KUKA KRL program: ap_15.src, ap_15.dat

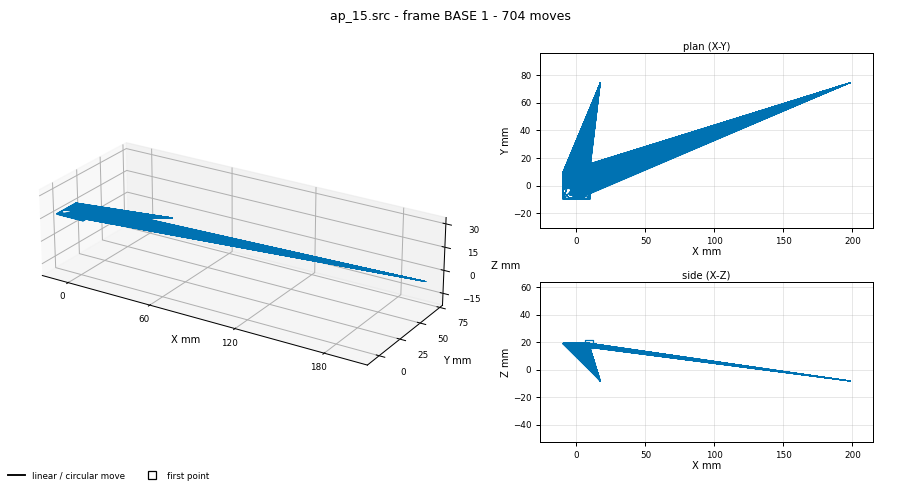
[picture p0: tool path of ap_15.src in frame BASE 1, 704 of 704 moves have a stored position in this frame; points joined in program order, loops and branches not executed]
--- ap_15.src ---
&ACCESS RVP
&REL 65
&PARAM DISKPATH = KRC:\R1\Program
DEF ap_15 ( )
   ;FOLD INI;%{PE}
     ;FOLD BASISTECH INI
       GLOBAL INTERRUPT DECL 3 WHEN $STOPMESS==TRUE DO IR_STOPM ( )
       INTERRUPT ON 3
       BAS (#INITMOV,0 )
     ;ENDFOLD (BASISTECH INI)
     ;FOLD USER INI
       ;Make your modifications here
     ;ENDFOLD (USER INI)
   ;ENDFOLD (INI)

   BAS (#VEL_PTP, 0020.0000)
   BAS (#ACC_PTP, 0020.0000)

   ;-----SET LIN AND ARC MOTION VARIABLES-----
   $VEL.ORI1 = 0350.0000
   $VEL.ORI2 = 0350.0000

   $ACC.CP = 0005.0000
   $ACC.ORI1 = 1000.0000
   $ACC.ORI2 = 1000.0000

   ;-----APPROXIMATION-----
   $APO.CVEL = 0100
   $APO.CPTP = 0100
   $APO.CDIS = 0006.0000
   $APO.CORI = 0090.0000

   BAS (#BASE, 1) ;Positioner
   BAS (#TOOL, 1) ;Vrashatel

   BAS(#VEL_PTP,15)                         ;;Set PTP Axis Velocity
   BAS(#ACC_PTP,50)                         ;;Set PTP Axis Acceleration
   PTP{A1 -92,A2 -133,A3 132,A4 7,A5 50,A6 -10}
   $VEL.CP = 0.060
   LIN  {X 9.039, Y 5.102, Z 18.500, A 0.000, B 0.000, C 0.000} C_DIS
   $VEL.CP = 0.060
   LIN  {X 9.040, Y 9.040, Z 18.500, A 0.000, B 0.000, C 0.000} C_DIS
   $VEL.CP = 0.060
   LIN  {X 9.039, Y 9.039, Z 18.500, A 0.000, B 0.000, C 0.000} C_DIS
   $VEL.CP = 0.060
   LIN  {X 4.069, Y 4.069, Z 18.500, A 0.000, B 0.000, C 0.000} C_DIS
   $VEL.CP = 0.060
   LIN  {X 3.708, Y 3.362, Z 18.500, A 0.000, B 0.000, C 0.000} C_DIS
   $VEL.CP = 0.060
   LIN  {X 9.039, Y -1.968, Z 18.500, A 0.000, B 0.000, C 0.000} C_DIS
   $VEL.CP = 0.060
   LIN  {X 9.039, Y 1.968, Z 18.500, A 0.000, B 0.000, C 0.000} C_DIS
   $VEL.CP = 0.060
   LIN  {X 3.551, Y -3.519, Z 18.500, A 0.000, B 0.000, C 0.000} C_DIS
   $VEL.CP = 0.060
   LIN  {X 0.185, Y -3.520, Z 18.500, A 0.000, B 0.000, C 0.000} C_DIS
   $VEL.CP = 0.060
   LIN  {X 1.313, Y -1.313, Z 18.500, A 0.000, B 0.000, C 0.000} C_DIS
   $VEL.CP = 0.060
   LIN  {X 3.519, Y -3.519, Z 18.500, A 0.000, B 0.000, C 0.000} C_DIS

;FOLD ARCOFF WDAT2 LIN P4 CPDAT2 Tool[1]:cmttorch Base[1]:vrashatel ;%{PE}
  ;FOLD Parameters ;%{h}
    ;Params IlfProvider=kukaroboter.arctech.arcofflin; Kuka.IsGlobalPoint=False; Kuka.PointName=P4; Kuka.BlendingEnabled=False; Kuka.MoveDataName=CPDAT2; Kuka.VelocityPath=0.01; Kuka.CurrentCDSetIndex=0; Kuka.MovementParameterFieldEnabled=True; ArcTech.WdatVarName=WDAT2; ArcTech.Basic=3.4.3.1264
  ;ENDFOLD
  $BWDSTART = FALSE
  LDAT_ACT = LCPDAT2
  FDAT_ACT = FP4
  BAS(#CP_PARAMS, gArcBasVelDefinition)
  SET_CD_PARAMS (0)
  TRIGGER WHEN PATH = ArcGetPath(#ArcOffBefore, WDAT2) DELAY = 0 DO ArcMainNG(#ArcOffBeforeOffStd, WDAT2, WP4) PRIO = -1
  TRIGGER WHEN PATH = ArcGetPath(#OnTheFlyArcOff, WDAT2) DELAY = 0 DO ArcMainNG(#ArcOffMoveStd, WDAT2, WP4) PRIO = -1
  ArcMainNG(#ArcOffBeforeMoveStd, WDAT2, WP4)
  LIN XP4
  ArcMainNG(#ArcOffAfterMoveStd, WDAT2, WP4)
;ENDFOLD
   $VEL.CP = 0.060
   LIN  {X 3.589, Y -3.589, Z 18.500, A 0.000, B 0.000, C 0.000} C_DIS
   $VEL.CP = 0.080
   LIN  {X 4.540, Y -4.052, Z 18.500, A 0.000, B 0.000, C 0.000} C_DIS
   $VEL.CP = 0.080
   LIN  {X 5.072, Y -6.953, Z 18.500, A 0.000, B 0.000, C 0.000} C_DIS

;FOLD ARCON WDAT1 LIN P3 Vel=0.5 m/s CPDAT1 Tool[1]:cmttorch Base[1]:vrashatel ;%{PE}
  ;FOLD Parameters ;%{h}
    ;Params IlfProvider=kukaroboter.arctech.arconlin; Kuka.IsGlobalPoint=False; Kuka.PointName=P3; Kuka.BlendingEnabled=False; Kuka.MoveDataName=CPDAT1; Kuka.VelocityPath=0.5; Kuka.CurrentCDSetIndex=0; Kuka.MovementParameterFieldEnabled=True; ArcTech.WdatVarName=WDAT1; ArcTech.Basic=3.4.3.1264
  ;ENDFOLD
  $BWDSTART = FALSE
  LDAT_ACT = LCPDAT1
  FDAT_ACT = FP3
  BAS(#CP_PARAMS, 0.5)
  SET_CD_PARAMS (0)
  TRIGGER WHEN DISTANCE = 1 DELAY = ArcGetDelay(#PreDefinition, WDAT1) DO ArcMainNG(#PreDefinition, WDAT1, WP3) PRIO = -1
  TRIGGER WHEN PATH = ArcGetPath(#OnTheFlyArcOn, WDAT1) DELAY = ArcGetDelay(#GasPreflow, WDAT1) DO ArcMainNG(#GasPreflow, WDAT1, WP3) PRIO = -1
  TRIGGER WHEN PATH = ArcGetPath(#OnTheFlyArcOn, WDAT1) DELAY = 0 DO ArcMainNG(#ArcOnMoveStd, WDAT1, WP3) PRIO = -1
  ArcMainNG(#ArcOnBeforeMoveStd, WDAT1, WP3)
  LIN XP3
  ArcMainNG(#ArcOnAfterMoveStd, WDAT1, WP3)
;ENDFOLD
   $VEL.CP = 0.060
   LIN  {X 5.071, Y -5.071, Z 18.500, A 0.000, B 0.000, C 0.000} C_DIS
   $VEL.CP = 0.060
   LIN  {X 9.039, Y -9.039, Z 18.500, A 0.000, B 0.000, C 0.000} C_DIS
   $VEL.CP = 0.060
   LIN  {X 9.039, Y -5.102, Z 18.500, A 0.000, B 0.000, C 0.000} C_DIS
   $VEL.CP = 0.060
   LIN  {X 5.102, Y -9.039, Z 18.500, A 0.000, B 0.000, C 0.000} C_DIS
   $VEL.CP = 0.060
   LIN  {X 1.968, Y -9.039, Z 18.500, A 0.000, B 0.000, C 0.000} C_DIS
   $VEL.CP = 0.060
   LIN  {X -0.118, Y -6.952, Z 18.500, A 0.000, B 0.000, C 0.000} C_DIS
   $VEL.CP = 0.060
   LIN  {X 0.118, Y -6.952, Z 18.500, A 0.000, B 0.000, C 0.000} C_DIS
   $VEL.CP = 0.060
   LIN  {X -1.968, Y -9.039, Z 18.500, A 0.000, B 0.000, C 0.000} C_DIS
   $VEL.CP = 0.060
   LIN  {X -5.102, Y -9.039, Z 18.500, A 0.000, B 0.000, C 0.000} C_DIS
   $VEL.CP = 0.060
   LIN  {X -9.039, Y -5.102, Z 18.500, A 0.000, B 0.000, C 0.000} C_DIS
   $VEL.CP = 0.060
   LIN  {X -9.039, Y -9.039, Z 18.500, A 0.000, B 0.000, C 0.000} C_DIS
   $VEL.CP = 0.060
   LIN  {X -3.903, Y -3.903, Z 18.500, A 0.000, B 0.000, C 0.000} C_DIS
   $VEL.CP = 0.060
   LIN  {X -3.655, Y -3.415, Z 18.500, A 0.000, B 0.000, C 0.000} C_DIS
   $VEL.CP = 0.060
   LIN  {X -9.039, Y 1.968, Z 18.500, A 0.000, B 0.000, C 0.000} C_DIS
   $VEL.CP = 0.060
   LIN  {X -9.039, Y -1.968, Z 18.500, A 0.000, B 0.000, C 0.000} C_DIS
   $VEL.CP = 0.060
   LIN  {X -3.226, Y 3.844, Z 18.500, A 0.000, B 0.000, C 0.000} C_DIS
   $VEL.CP = 0.060
   LIN  {X 0.049, Y 3.845, Z 18.500, A 0.000, B 0.000, C 0.000} C_DIS
   $VEL.CP = 0.060
   LIN  {X -1.267, Y 1.267, Z 18.500, A 0.000, B 0.000, C 0.000} C_DIS
   $VEL.CP = 0.060
   LIN  {X -3.844, Y 3.844, Z 18.500, A 0.000, B 0.000, C 0.000} C_DIS
   $VEL.CP = 0.060
   LIN  {X -4.554, Y 3.845, Z 18.500, A 0.000, B 0.000, C 0.000} C_DIS
   $VEL.CP = 0.060
   LIN  {X -4.553, Y 4.553, Z 18.500, A 0.000, B 0.000, C 0.000} C_DIS
   $VEL.CP = 0.060
   LIN  {X -9.039, Y 9.039, Z 18.500, A 0.000, B 0.000, C 0.000} C_DIS
   $VEL.CP = 0.060
   LIN  {X -9.040, Y 9.040, Z 18.500, A 0.000, B 0.000, C 0.000} C_DIS

;FOLD ARCOFF WDAT2 LIN P4 CPDAT2 Tool[1]:cmttorch Base[1]:vrashatel ;%{PE}
  ;FOLD Parameters ;%{h}
    ;Params IlfProvider=kukaroboter.arctech.arcofflin; Kuka.IsGlobalPoint=False; Kuka.PointName=P4; Kuka.BlendingEnabled=False; Kuka.MoveDataName=CPDAT2; Kuka.VelocityPath=0.01; Kuka.CurrentCDSetIndex=0; Kuka.MovementParameterFieldEnabled=True; ArcTech.WdatVarName=WDAT2; ArcTech.Basic=3.4.3.1264
  ;ENDFOLD
  $BWDSTART = FALSE
  LDAT_ACT = LCPDAT2
  FDAT_ACT = FP4
  BAS(#CP_PARAMS, gArcBasVelDefinition)
  SET_CD_PARAMS (0)
  TRIGGER WHEN PATH = ArcGetPath(#ArcOffBefore, WDAT2) DELAY = 0 DO ArcMainNG(#ArcOffBeforeOffStd, WDAT2, WP4) PRIO = -1
  TRIGGER WHEN PATH = ArcGetPath(#OnTheFlyArcOff, WDAT2) DELAY = 0 DO ArcMainNG(#ArcOffMoveStd, WDAT2, WP4) PRIO = -1
  ArcMainNG(#ArcOffBeforeMoveStd, WDAT2, WP4)
  LIN XP4
  ArcMainNG(#ArcOffAfterMoveStd, WDAT2, WP4)
;ENDFOLD
   $VEL.CP = 0.010
   LIN  {X -9.040, Y 9.040, Z 18.700, A 0.000, B 0.000, C 0.000} C_DIS
   $VEL.CP = 0.080
   LIN  {X -9.530, Y 9.530, Z 18.700, A 0.000, B 0.000, C 0.000} C_DIS
   $VEL.CP = 0.080
   LIN  {X -9.800, Y 9.800, Z 18.700, A 0.000, B 0.000, C 0.000} C_DIS

;FOLD ARCON WDAT1 LIN P3 Vel=0.5 m/s CPDAT1 Tool[1]:cmttorch Base[1]:vrashatel ;%{PE}
  ;FOLD Parameters ;%{h}
    ;Params IlfProvider=kukaroboter.arctech.arconlin; Kuka.IsGlobalPoint=False; Kuka.PointName=P3; Kuka.BlendingEnabled=False; Kuka.MoveDataName=CPDAT1; Kuka.VelocityPath=0.5; Kuka.CurrentCDSetIndex=0; Kuka.MovementParameterFieldEnabled=True; ArcTech.WdatVarName=WDAT1; ArcTech.Basic=3.4.3.1264
  ;ENDFOLD
  $BWDSTART = FALSE
  LDAT_ACT = LCPDAT1
  FDAT_ACT = FP3
  BAS(#CP_PARAMS, 0.5)
  SET_CD_PARAMS (0)
  TRIGGER WHEN DISTANCE = 1 DELAY = ArcGetDelay(#PreDefinition, WDAT1) DO ArcMainNG(#PreDefinition, WDAT1, WP3) PRIO = -1
  TRIGGER WHEN PATH = ArcGetPath(#OnTheFlyArcOn, WDAT1) DELAY = ArcGetDelay(#GasPreflow, WDAT1) DO ArcMainNG(#GasPreflow, WDAT1, WP3) PRIO = -1
  TRIGGER WHEN PATH = ArcGetPath(#OnTheFlyArcOn, WDAT1) DELAY = 0 DO ArcMainNG(#ArcOnMoveStd, WDAT1, WP3) PRIO = -1
  ArcMainNG(#ArcOnBeforeMoveStd, WDAT1, WP3)
  LIN XP3
  ArcMainNG(#ArcOnAfterMoveStd, WDAT1, WP3)
;ENDFOLD
   $VEL.CP = 0.025
   LIN  {X -9.800, Y 9.800, Z 18.700, A 0.000, B 0.000, C 0.000} C_DIS
   $VEL.CP = 0.060
   LIN  {X -9.800, Y -9.800, Z 18.700, A 0.000, B 0.000, C 0.000} C_DIS
   $VEL.CP = 0.060
   LIN  {X 9.800, Y -9.800, Z 18.700, A 0.000, B 0.000, C 0.000} C_DIS
   $VEL.CP = 0.060
   LIN  {X 9.800, Y 9.800, Z 18.700, A 0.000, B 0.000, C 0.000} C_DIS
   $VEL.CP = 0.060
   LIN  {X -9.800, Y 9.800, Z 18.700, A 0.000, B 0.000, C 0.000} C_DIS

;FOLD ARCOFF WDAT2 LIN P4 CPDAT2 Tool[1]:cmttorch Base[1]:vrashatel ;%{PE}
  ;FOLD Parameters ;%{h}
    ;Params IlfProvider=kukaroboter.arctech.arcofflin; Kuka.IsGlobalPoint=False; Kuka.PointName=P4; Kuka.BlendingEnabled=False; Kuka.MoveDataName=CPDAT2; Kuka.VelocityPath=0.01; Kuka.CurrentCDSetIndex=0; Kuka.MovementParameterFieldEnabled=True; ArcTech.WdatVarName=WDAT2; ArcTech.Basic=3.4.3.1264
  ;ENDFOLD
  $BWDSTART = FALSE
  LDAT_ACT = LCPDAT2
  FDAT_ACT = FP4
  BAS(#CP_PARAMS, gArcBasVelDefinition)
  SET_CD_PARAMS (0)
  TRIGGER WHEN PATH = ArcGetPath(#ArcOffBefore, WDAT2) DELAY = 0 DO ArcMainNG(#ArcOffBeforeOffStd, WDAT2, WP4) PRIO = -1
  TRIGGER WHEN PATH = ArcGetPath(#OnTheFlyArcOff, WDAT2) DELAY = 0 DO ArcMainNG(#ArcOffMoveStd, WDAT2, WP4) PRIO = -1
  ArcMainNG(#ArcOffBeforeMoveStd, WDAT2, WP4)
  LIN XP4
  ArcMainNG(#ArcOffAfterMoveStd, WDAT2, WP4)
;ENDFOLD
   $VEL.CP = 0.080
   LIN  {X -9.800, Y 9.600, Z 18.700, A 0.000, B 0.000, C 0.000} C_DIS
   $VEL.CP = 0.080
   LIN  {X -9.360, Y 9.360, Z 18.700, A 0.000, B 0.000, C 0.000} C_DIS
   $VEL.CP = 0.080
   LIN  {X -4.094, Y 4.605, Z 18.700, A 0.000, B 0.000, C 0.000} C_DIS
   $VEL.CP = 0.080
   LIN  {X -3.794, Y 4.605, Z 18.700, A 0.000, B 0.000, C 0.000} C_DIS

;FOLD ARCON WDAT1 LIN P3 Vel=0.5 m/s CPDAT1 Tool[1]:cmttorch Base[1]:vrashatel ;%{PE}
  ;FOLD Parameters ;%{h}
    ;Params IlfProvider=kukaroboter.arctech.arconlin; Kuka.IsGlobalPoint=False; Kuka.PointName=P3; Kuka.BlendingEnabled=False; Kuka.MoveDataName=CPDAT1; Kuka.VelocityPath=0.5; Kuka.CurrentCDSetIndex=0; Kuka.MovementParameterFieldEnabled=True; ArcTech.WdatVarName=WDAT1; ArcTech.Basic=3.4.3.1264
  ;ENDFOLD
  $BWDSTART = FALSE
  LDAT_ACT = LCPDAT1
  FDAT_ACT = FP3
  BAS(#CP_PARAMS, 0.5)
  SET_CD_PARAMS (0)
  TRIGGER WHEN DISTANCE = 1 DELAY = ArcGetDelay(#PreDefinition, WDAT1) DO ArcMainNG(#PreDefinition, WDAT1, WP3) PRIO = -1
  TRIGGER WHEN PATH = ArcGetPath(#OnTheFlyArcOn, WDAT1) DELAY = ArcGetDelay(#GasPreflow, WDAT1) DO ArcMainNG(#GasPreflow, WDAT1, WP3) PRIO = -1
  TRIGGER WHEN PATH = ArcGetPath(#OnTheFlyArcOn, WDAT1) DELAY = 0 DO ArcMainNG(#ArcOnMoveStd, WDAT1, WP3) PRIO = -1
  ArcMainNG(#ArcOnBeforeMoveStd, WDAT1, WP3)
  LIN XP3
  ArcMainNG(#ArcOnAfterMoveStd, WDAT1, WP3)
;ENDFOLD
   $VEL.CP = 0.060
   LIN  {X -3.794, Y 6.518, Z 18.700, A 0.000, B 0.000, C 0.000} C_DIS
   $VEL.CP = 0.060
   LIN  {X 4.127, Y 6.518, Z 18.700, A 0.000, B 0.000, C 0.000} C_DIS
   $VEL.CP = 0.060
   LIN  {X 4.127, Y 5.850, Z 18.700, A 0.000, B 0.000, C 0.000} C_DIS
   $VEL.CP = 0.060
   LIN  {X -1.057, Y -4.280, Z 18.700, A 0.000, B 0.000, C 0.000} C_DIS
   $VEL.CP = 0.060
   LIN  {X 4.312, Y -4.280, Z 18.700, A 0.000, B 0.000, C 0.000} C_DIS
   $VEL.CP = 0.060
   LIN  {X 4.312, Y -6.193, Z 18.700, A 0.000, B 0.000, C 0.000} C_DIS
   $VEL.CP = 0.060
   LIN  {X -3.878, Y -6.193, Z 18.700, A 0.000, B 0.000, C 0.000} C_DIS
   $VEL.CP = 0.060
   LIN  {X -3.878, Y -5.525, Z 18.700, A 0.000, B 0.000, C 0.000} C_DIS
   $VEL.CP = 0.060
   LIN  {X 1.290, Y 4.605, Z 18.700, A 0.000, B 0.000, C 0.000} C_DIS
   $VEL.CP = 0.060
   LIN  {X -3.794, Y 4.605, Z 18.700, A 0.000, B 0.000, C 0.000} C_DIS

;FOLD ARCOFF WDAT2 LIN P4 CPDAT2 Tool[1]:cmttorch Base[1]:vrashatel ;%{PE}
  ;FOLD Parameters ;%{h}
    ;Params IlfProvider=kukaroboter.arctech.arcofflin; Kuka.IsGlobalPoint=False; Kuka.PointName=P4; Kuka.BlendingEnabled=False; Kuka.MoveDataName=CPDAT2; Kuka.VelocityPath=0.01; Kuka.CurrentCDSetIndex=0; Kuka.MovementParameterFieldEnabled=True; ArcTech.WdatVarName=WDAT2; ArcTech.Basic=3.4.3.1264
  ;ENDFOLD
  $BWDSTART = FALSE
  LDAT_ACT = LCPDAT2
  FDAT_ACT = FP4
  BAS(#CP_PARAMS, gArcBasVelDefinition)
  SET_CD_PARAMS (0)
  TRIGGER WHEN PATH = ArcGetPath(#ArcOffBefore, WDAT2) DELAY = 0 DO ArcMainNG(#ArcOffBeforeOffStd, WDAT2, WP4) PRIO = -1
  TRIGGER WHEN PATH = ArcGetPath(#OnTheFlyArcOff, WDAT2) DELAY = 0 DO ArcMainNG(#ArcOffMoveStd, WDAT2, WP4) PRIO = -1
  ArcMainNG(#ArcOffBeforeMoveStd, WDAT2, WP4)
  LIN XP4
  ArcMainNG(#ArcOffAfterMoveStd, WDAT2, WP4)
;ENDFOLD
   $VEL.CP = 0.080
   LIN  {X -3.794, Y 4.805, Z 18.700, A 0.000, B 0.000, C 0.000} C_DIS
   $VEL.CP = 0.080
   LIN  {X -4.194, Y 4.205, Z 18.700, A 0.000, B 0.000, C 0.000} C_DIS

;FOLD ARCON WDAT1 LIN P3 Vel=0.5 m/s CPDAT1 Tool[1]:cmttorch Base[1]:vrashatel ;%{PE}
  ;FOLD Parameters ;%{h}
    ;Params IlfProvider=kukaroboter.arctech.arconlin; Kuka.IsGlobalPoint=False; Kuka.PointName=P3; Kuka.BlendingEnabled=False; Kuka.MoveDataName=CPDAT1; Kuka.VelocityPath=0.5; Kuka.CurrentCDSetIndex=0; Kuka.MovementParameterFieldEnabled=True; ArcTech.WdatVarName=WDAT1; ArcTech.Basic=3.4.3.1264
  ;ENDFOLD
  $BWDSTART = FALSE
  LDAT_ACT = LCPDAT1
  FDAT_ACT = FP3
  BAS(#CP_PARAMS, 0.5)
  SET_CD_PARAMS (0)
  TRIGGER WHEN DISTANCE = 1 DELAY = ArcGetDelay(#PreDefinition, WDAT1) DO ArcMainNG(#PreDefinition, WDAT1, WP3) PRIO = -1
  TRIGGER WHEN PATH = ArcGetPath(#OnTheFlyArcOn, WDAT1) DELAY = ArcGetDelay(#GasPreflow, WDAT1) DO ArcMainNG(#GasPreflow, WDAT1, WP3) PRIO = -1
  TRIGGER WHEN PATH = ArcGetPath(#OnTheFlyArcOn, WDAT1) DELAY = 0 DO ArcMainNG(#ArcOnMoveStd, WDAT1, WP3) PRIO = -1
  ArcMainNG(#ArcOnBeforeMoveStd, WDAT1, WP3)
  LIN XP3
  ArcMainNG(#ArcOnAfterMoveStd, WDAT1, WP3)
;ENDFOLD
   $VEL.CP = 0.060
   LIN  {X -4.194, Y 6.918, Z 18.700, A 0.000, B 0.000, C 0.000} C_DIS
   $VEL.CP = 0.060
   LIN  {X 4.527, Y 6.918, Z 18.700, A 0.000, B 0.000, C 0.000} C_DIS
   $VEL.CP = 0.060
   LIN  {X 4.527, Y 5.754, Z 18.700, A 0.000, B 0.000, C 0.000} C_DIS
   $VEL.CP = 0.060
   LIN  {X -0.403, Y -3.880, Z 18.700, A 0.000, B 0.000, C 0.000} C_DIS
   $VEL.CP = 0.060
   LIN  {X 4.712, Y -3.880, Z 18.700, A 0.000, B 0.000, C 0.000} C_DIS
   $VEL.CP = 0.060
   LIN  {X 4.712, Y -6.593, Z 18.700, A 0.000, B 0.000, C 0.000} C_DIS
   $VEL.CP = 0.060
   LIN  {X -4.278, Y -6.593, Z 18.700, A 0.000, B 0.000, C 0.000} C_DIS
   $VEL.CP = 0.060
   LIN  {X -4.278, Y -5.429, Z 18.700, A 0.000, B 0.000, C 0.000} C_DIS
   $VEL.CP = 0.060
   LIN  {X 0.637, Y 4.205, Z 18.700, A 0.000, B 0.000, C 0.000} C_DIS
   $VEL.CP = 0.060
   LIN  {X -4.194, Y 4.205, Z 18.700, A 0.000, B 0.000, C 0.000} C_DIS

;FOLD ARCOFF WDAT2 LIN P4 CPDAT2 Tool[1]:cmttorch Base[1]:vrashatel ;%{PE}
  ;FOLD Parameters ;%{h}
    ;Params IlfProvider=kukaroboter.arctech.arcofflin; Kuka.IsGlobalPoint=False; Kuka.PointName=P4; Kuka.BlendingEnabled=False; Kuka.MoveDataName=CPDAT2; Kuka.VelocityPath=0.01; Kuka.CurrentCDSetIndex=0; Kuka.MovementParameterFieldEnabled=True; ArcTech.WdatVarName=WDAT2; ArcTech.Basic=3.4.3.1264
  ;ENDFOLD
  $BWDSTART = FALSE
  LDAT_ACT = LCPDAT2
  FDAT_ACT = FP4
  BAS(#CP_PARAMS, gArcBasVelDefinition)
  SET_CD_PARAMS (0)
  TRIGGER WHEN PATH = ArcGetPath(#ArcOffBefore, WDAT2) DELAY = 0 DO ArcMainNG(#ArcOffBeforeOffStd, WDAT2, WP4) PRIO = -1
  TRIGGER WHEN PATH = ArcGetPath(#OnTheFlyArcOff, WDAT2) DELAY = 0 DO ArcMainNG(#ArcOffMoveStd, WDAT2, WP4) PRIO = -1
  ArcMainNG(#ArcOffBeforeMoveStd, WDAT2, WP4)
  LIN XP4
  ArcMainNG(#ArcOffAfterMoveStd, WDAT2, WP4)
;ENDFOLD
   $VEL.CP = 0.080
   LIN  {X -9.400, Y 9.400, Z 18.700, A 0.000, B 0.000, C 0.000} C_DIS

;FOLD ARCON WDAT1 LIN P3 Vel=0.5 m/s CPDAT1 Tool[1]:cmttorch Base[1]:vrashatel ;%{PE}
  ;FOLD Parameters ;%{h}
    ;Params IlfProvider=kukaroboter.arctech.arconlin; Kuka.IsGlobalPoint=False; Kuka.PointName=P3; Kuka.BlendingEnabled=False; Kuka.MoveDataName=CPDAT1; Kuka.VelocityPath=0.5; Kuka.CurrentCDSetIndex=0; Kuka.MovementParameterFieldEnabled=True; ArcTech.WdatVarName=WDAT1; ArcTech.Basic=3.4.3.1264
  ;ENDFOLD
  $BWDSTART = FALSE
  LDAT_ACT = LCPDAT1
  FDAT_ACT = FP3
  BAS(#CP_PARAMS, 0.5)
  SET_CD_PARAMS (0)
  TRIGGER WHEN DISTANCE = 1 DELAY = ArcGetDelay(#PreDefinition, WDAT1) DO ArcMainNG(#PreDefinition, WDAT1, WP3) PRIO = -1
  TRIGGER WHEN PATH = ArcGetPath(#OnTheFlyArcOn, WDAT1) DELAY = ArcGetDelay(#GasPreflow, WDAT1) DO ArcMainNG(#GasPreflow, WDAT1, WP3) PRIO = -1
  TRIGGER WHEN PATH = ArcGetPath(#OnTheFlyArcOn, WDAT1) DELAY = 0 DO ArcMainNG(#ArcOnMoveStd, WDAT1, WP3) PRIO = -1
  ArcMainNG(#ArcOnBeforeMoveStd, WDAT1, WP3)
  LIN XP3
  ArcMainNG(#ArcOnAfterMoveStd, WDAT1, WP3)
;ENDFOLD
   $VEL.CP = 0.060
   LIN  {X -9.400, Y -9.400, Z 18.700, A 0.000, B 0.000, C 0.000} C_DIS
   $VEL.CP = 0.060
   LIN  {X 9.400, Y -9.400, Z 18.700, A 0.000, B 0.000, C 0.000} C_DIS
   $VEL.CP = 0.060
   LIN  {X 9.400, Y 9.400, Z 18.700, A 0.000, B 0.000, C 0.000} C_DIS
   $VEL.CP = 0.060
   LIN  {X -9.400, Y 9.400, Z 18.700, A 0.000, B 0.000, C 0.000} C_DIS

;FOLD ARCOFF WDAT2 LIN P4 CPDAT2 Tool[1]:cmttorch Base[1]:vrashatel ;%{PE}
  ;FOLD Parameters ;%{h}
    ;Params IlfProvider=kukaroboter.arctech.arcofflin; Kuka.IsGlobalPoint=False; Kuka.PointName=P4; Kuka.BlendingEnabled=False; Kuka.MoveDataName=CPDAT2; Kuka.VelocityPath=0.01; Kuka.CurrentCDSetIndex=0; Kuka.MovementParameterFieldEnabled=True; ArcTech.WdatVarName=WDAT2; ArcTech.Basic=3.4.3.1264
  ;ENDFOLD
  $BWDSTART = FALSE
  LDAT_ACT = LCPDAT2
  FDAT_ACT = FP4
  BAS(#CP_PARAMS, gArcBasVelDefinition)
  SET_CD_PARAMS (0)
  TRIGGER WHEN PATH = ArcGetPath(#ArcOffBefore, WDAT2) DELAY = 0 DO ArcMainNG(#ArcOffBeforeOffStd, WDAT2, WP4) PRIO = -1
  TRIGGER WHEN PATH = ArcGetPath(#OnTheFlyArcOff, WDAT2) DELAY = 0 DO ArcMainNG(#ArcOffMoveStd, WDAT2, WP4) PRIO = -1
  ArcMainNG(#ArcOffBeforeMoveStd, WDAT2, WP4)
  LIN XP4
  ArcMainNG(#ArcOffAfterMoveStd, WDAT2, WP4)
;ENDFOLD
   $VEL.CP = 0.080
   LIN  {X -9.040, Y 9.040, Z 18.700, A 0.000, B 0.000, C 0.000} C_DIS

;FOLD ARCON WDAT1 LIN P3 Vel=0.5 m/s CPDAT1 Tool[1]:cmttorch Base[1]:vrashatel ;%{PE}
  ;FOLD Parameters ;%{h}
    ;Params IlfProvider=kukaroboter.arctech.arconlin; Kuka.IsGlobalPoint=False; Kuka.PointName=P3; Kuka.BlendingEnabled=False; Kuka.MoveDataName=CPDAT1; Kuka.VelocityPath=0.5; Kuka.CurrentCDSetIndex=0; Kuka.MovementParameterFieldEnabled=True; ArcTech.WdatVarName=WDAT1; ArcTech.Basic=3.4.3.1264
  ;ENDFOLD
  $BWDSTART = FALSE
  LDAT_ACT = LCPDAT1
  FDAT_ACT = FP3
  BAS(#CP_PARAMS, 0.5)
  SET_CD_PARAMS (0)
  TRIGGER WHEN DISTANCE = 1 DELAY = ArcGetDelay(#PreDefinition, WDAT1) DO ArcMainNG(#PreDefinition, WDAT1, WP3) PRIO = -1
  TRIGGER WHEN PATH = ArcGetPath(#OnTheFlyArcOn, WDAT1) DELAY = ArcGetDelay(#GasPreflow, WDAT1) DO ArcMainNG(#GasPreflow, WDAT1, WP3) PRIO = -1
  TRIGGER WHEN PATH = ArcGetPath(#OnTheFlyArcOn, WDAT1) DELAY = 0 DO ArcMainNG(#ArcOnMoveStd, WDAT1, WP3) PRIO = -1
  ArcMainNG(#ArcOnBeforeMoveStd, WDAT1, WP3)
  LIN XP3
  ArcMainNG(#ArcOnAfterMoveStd, WDAT1, WP3)
;ENDFOLD
   $VEL.CP = 0.060
   LIN  {X -9.039, Y 5.102, Z 18.700, A 0.000, B 0.000, C 0.000} C_DIS
   $VEL.CP = 0.060
   LIN  {X -5.102, Y 9.039, Z 18.700, A 0.000, B 0.000, C 0.000} C_DIS
   $VEL.CP = 0.060
   LIN  {X -1.968, Y 9.039, Z 18.700, A 0.000, B 0.000, C 0.000} C_DIS
   $VEL.CP = 0.060
   LIN  {X -0.205, Y 7.276, Z 18.700, A 0.000, B 0.000, C 0.000} C_DIS
   $VEL.CP = 0.060
   LIN  {X 0.206, Y 7.277, Z 18.700, A 0.000, B 0.000, C 0.000} C_DIS
   $VEL.CP = 0.060
   LIN  {X 1.968, Y 9.039, Z 18.700, A 0.000, B 0.000, C 0.000} C_DIS
   $VEL.CP = 0.060
   LIN  {X 5.102, Y 9.039, Z 18.700, A 0.000, B 0.000, C 0.000} C_DIS
   $VEL.CP = 0.060
   LIN  {X 9.039, Y 5.102, Z 18.700, A 0.000, B 0.000, C 0.000} C_DIS
   $VEL.CP = 0.060
   LIN  {X 9.040, Y 9.040, Z 18.700, A 0.000, B 0.000, C 0.000} C_DIS
   $VEL.CP = 0.060
   LIN  {X 9.039, Y 9.039, Z 18.700, A 0.000, B 0.000, C 0.000} C_DIS
   $VEL.CP = 0.060
   LIN  {X 4.069, Y 4.069, Z 18.700, A 0.000, B 0.000, C 0.000} C_DIS
   $VEL.CP = 0.060
   LIN  {X 3.708, Y 3.362, Z 18.700, A 0.000, B 0.000, C 0.000} C_DIS
   $VEL.CP = 0.060
   LIN  {X 9.039, Y -1.968, Z 18.700, A 0.000, B 0.000, C 0.000} C_DIS
   $VEL.CP = 0.060
   LIN  {X 9.039, Y 1.968, Z 18.700, A 0.000, B 0.000, C 0.000} C_DIS
   $VEL.CP = 0.060
   LIN  {X 3.551, Y -3.519, Z 18.700, A 0.000, B 0.000, C 0.000} C_DIS
   $VEL.CP = 0.060
   LIN  {X 0.185, Y -3.520, Z 18.700, A 0.000, B 0.000, C 0.000} C_DIS
   $VEL.CP = 0.060
   LIN  {X 1.313, Y -1.313, Z 18.700, A 0.000, B 0.000, C 0.000} C_DIS
   $VEL.CP = 0.060
   LIN  {X 3.519, Y -3.519, Z 18.700, A 0.000, B 0.000, C 0.000} C_DIS

;FOLD ARCOFF WDAT2 LIN P4 CPDAT2 Tool[1]:cmttorch Base[1]:vrashatel ;%{PE}
  ;FOLD Parameters ;%{h}
    ;Params IlfProvider=kukaroboter.arctech.arcofflin; Kuka.IsGlobalPoint=False; Kuka.PointName=P4; Kuka.BlendingEnabled=False; Kuka.MoveDataName=CPDAT2; Kuka.VelocityPath=0.01; Kuka.CurrentCDSetIndex=0; Kuka.MovementParameterFieldEnabled=True; ArcTech.WdatVarName=WDAT2; ArcTech.Basic=3.4.3.1264
  ;ENDFOLD
  $BWDSTART = FALSE
  LDAT_ACT = LCPDAT2
  FDAT_ACT = FP4
  BAS(#CP_PARAMS, gArcBasVelDefinition)
  SET_CD_PARAMS (0)
  TRIGGER WHEN PATH = ArcGetPath(#ArcOffBefore, WDAT2) DELAY = 0 DO ArcMainNG(#ArcOffBeforeOffStd, WDAT2, WP4) PRIO = -1
  TRIGGER WHEN PATH = ArcGetPath(#OnTheFlyArcOff, WDAT2) DELAY = 0 DO ArcMainNG(#ArcOffMoveStd, WDAT2, WP4) PRIO = -1
  ArcMainNG(#ArcOffBeforeMoveStd, WDAT2, WP4)
  LIN XP4
  ArcMainNG(#ArcOffAfterMoveStd, WDAT2, WP4)
;ENDFOLD
   $VEL.CP = 0.060
   LIN  {X 3.589, Y -3.589, Z 18.700, A 0.000, B 0.000, C 0.000} C_DIS
   $VEL.CP = 0.080
   LIN  {X 4.540, Y -4.052, Z 18.700, A 0.000, B 0.000, C 0.000} C_DIS
   $VEL.CP = 0.080
   LIN  {X 5.072, Y -6.953, Z 18.700, A 0.000, B 0.000, C 0.000} C_DIS

;FOLD ARCON WDAT1 LIN P3 Vel=0.5 m/s CPDAT1 Tool[1]:cmttorch Base[1]:vrashatel ;%{PE}
  ;FOLD Parameters ;%{h}
    ;Params IlfProvider=kukaroboter.arctech.arconlin; Kuka.IsGlobalPoint=False; Kuka.PointName=P3; Kuka.BlendingEnabled=False; Kuka.MoveDataName=CPDAT1; Kuka.VelocityPath=0.5; Kuka.CurrentCDSetIndex=0; Kuka.MovementParameterFieldEnabled=True; ArcTech.WdatVarName=WDAT1; ArcTech.Basic=3.4.3.1264
  ;ENDFOLD
  $BWDSTART = FALSE
  LDAT_ACT = LCPDAT1
  FDAT_ACT = FP3
  BAS(#CP_PARAMS, 0.5)
  SET_CD_PARAMS (0)
  TRIGGER WHEN DISTANCE = 1 DELAY = ArcGetDelay(#PreDefinition, WDAT1) DO ArcMainNG(#PreDefinition, WDAT1, WP3) PRIO = -1
  TRIGGER WHEN PATH = ArcGetPath(#OnTheFlyArcOn, WDAT1) DELAY = ArcGetDelay(#GasPreflow, WDAT1) DO ArcMainNG(#GasPreflow, WDAT1, WP3) PRIO = -1
  TRIGGER WHEN PATH = ArcGetPath(#OnTheFlyArcOn, WDAT1) DELAY = 0 DO ArcMainNG(#ArcOnMoveStd, WDAT1, WP3) PRIO = -1
  ArcMainNG(#ArcOnBeforeMoveStd, WDAT1, WP3)
  LIN XP3
  ArcMainNG(#ArcOnAfterMoveStd, WDAT1, WP3)
;ENDFOLD
   $VEL.CP = 0.060
   LIN  {X 5.071, Y -5.071, Z 18.700, A 0.000, B 0.000, C 0.000} C_DIS
   $VEL.CP = 0.060
   LIN  {X 9.039, Y -9.039, Z 18.700, A 0.000, B 0.000, C 0.000} C_DIS
   $VEL.CP = 0.060
   LIN  {X 9.039, Y -5.102, Z 18.700, A 0.000, B 0.000, C 0.000} C_DIS
   $VEL.CP = 0.060
   LIN  {X 5.102, Y -9.039, Z 18.700, A 0.000, B 0.000, C 0.000} C_DIS
   $VEL.CP = 0.060
   LIN  {X 1.968, Y -9.039, Z 18.700, A 0.000, B 0.000, C 0.000} C_DIS
   $VEL.CP = 0.060
   LIN  {X -0.118, Y -6.952, Z 18.700, A 0.000, B 0.000, C 0.000} C_DIS
   $VEL.CP = 0.060
   LIN  {X 0.118, Y -6.952, Z 18.700, A 0.000, B 0.000, C 0.000} C_DIS
   $VEL.CP = 0.060
   LIN  {X -1.968, Y -9.039, Z 18.700, A 0.000, B 0.000, C 0.000} C_DIS
   $VEL.CP = 0.060
   LIN  {X -5.102, Y -9.039, Z 18.700, A 0.000, B 0.000, C 0.000} C_DIS
   $VEL.CP = 0.060
   LIN  {X -9.039, Y -5.102, Z 18.700, A 0.000, B 0.000, C 0.000} C_DIS
   $VEL.CP = 0.060
   LIN  {X -9.039, Y -9.039, Z 18.700, A 0.000, B 0.000, C 0.000} C_DIS
   $VEL.CP = 0.060
   LIN  {X -3.903, Y -3.903, Z 18.700, A 0.000, B 0.000, C 0.000} C_DIS
   $VEL.CP = 0.060
   LIN  {X -3.655, Y -3.415, Z 18.700, A 0.000, B 0.000, C 0.000} C_DIS
   $VEL.CP = 0.060
   LIN  {X -9.039, Y 1.968, Z 18.700, A 0.000, B 0.000, C 0.000} C_DIS
   $VEL.CP = 0.060
   LIN  {X -9.039, Y -1.968, Z 18.700, A 0.000, B 0.000, C 0.000} C_DIS
   $VEL.CP = 0.060
   LIN  {X -3.226, Y 3.844, Z 18.700, A 0.000, B 0.000, C 0.000} C_DIS
   $VEL.CP = 0.060
   LIN  {X 0.049, Y 3.845, Z 18.700, A 0.000, B 0.000, C 0.000} C_DIS
   $VEL.CP = 0.060
   LIN  {X -1.267, Y 1.267, Z 18.700, A 0.000, B 0.000, C 0.000} C_DIS
   $VEL.CP = 0.060
   LIN  {X -3.844, Y 3.844, Z 18.700, A 0.000, B 0.000, C 0.000} C_DIS
   $VEL.CP = 0.060
   LIN  {X -4.554, Y 3.845, Z 18.700, A 0.000, B 0.000, C 0.000} C_DIS
   $VEL.CP = 0.060
   LIN  {X -4.553, Y 4.553, Z 18.700, A 0.000, B 0.000, C 0.000} C_DIS
   $VEL.CP = 0.060
   LIN  {X -9.039, Y 9.039, Z 18.700, A 0.000, B 0.000, C 0.000} C_DIS
   $VEL.CP = 0.060
   LIN  {X -9.040, Y 9.040, Z 18.700, A 0.000, B 0.000, C 0.000} C_DIS

;FOLD ARCOFF WDAT2 LIN P4 CPDAT2 Tool[1]:cmttorch Base[1]:vrashatel ;%{PE}
  ;FOLD Parameters ;%{h}
    ;Params IlfProvider=kukaroboter.arctech.arcofflin; Kuka.IsGlobalPoint=False; Kuka.PointName=P4; Kuka.BlendingEnabled=False; Kuka.MoveDataName=CPDAT2; Kuka.VelocityPath=0.01; Kuka.CurrentCDSetIndex=0; Kuka.MovementParameterFieldEnabled=True; ArcTech.WdatVarName=WDAT2; ArcTech.Basic=3.4.3.1264
  ;ENDFOLD
  $BWDSTART = FALSE
  LDAT_ACT = LCPDAT2
  FDAT_ACT = FP4
  BAS(#CP_PARAMS, gArcBasVelDefinition)
  SET_CD_PARAMS (0)
  TRIGGER WHEN PATH = ArcGetPath(#ArcOffBefore, WDAT2) DELAY = 0 DO ArcMainNG(#ArcOffBeforeOffStd, WDAT2, WP4) PRIO = -1
  TRIGGER WHEN PATH = ArcGetPath(#OnTheFlyArcOff, WDAT2) DELAY = 0 DO ArcMainNG(#ArcOffMoveStd, WDAT2, WP4) PRIO = -1
  ArcMainNG(#ArcOffBeforeMoveStd, WDAT2, WP4)
  LIN XP4
  ArcMainNG(#ArcOffAfterMoveStd, WDAT2, WP4)
;ENDFOLD
   $VEL.CP = 0.010
   LIN  {X -9.040, Y 9.040, Z 18.900, A 0.000, B 0.000, C 0.000} C_DIS
   $VEL.CP = 0.080
   LIN  {X -9.530, Y 9.530, Z 18.900, A 0.000, B 0.000, C 0.000} C_DIS
   $VEL.CP = 0.080
   LIN  {X -9.800, Y 9.800, Z 18.900, A 0.000, B 0.000, C 0.000} C_DIS

;FOLD ARCON WDAT1 LIN P3 Vel=0.5 m/s CPDAT1 Tool[1]:cmttorch Base[1]:vrashatel ;%{PE}
  ;FOLD Parameters ;%{h}
    ;Params IlfProvider=kukaroboter.arctech.arconlin; Kuka.IsGlobalPoint=False; Kuka.PointName=P3; Kuka.BlendingEnabled=False; Kuka.MoveDataName=CPDAT1; Kuka.VelocityPath=0.5; Kuka.CurrentCDSetIndex=0; Kuka.MovementParameterFieldEnabled=True; ArcTech.WdatVarName=WDAT1; ArcTech.Basic=3.4.3.1264
  ;ENDFOLD
  $BWDSTART = FALSE
  LDAT_ACT = LCPDAT1
  FDAT_ACT = FP3
  BAS(#CP_PARAMS, 0.5)
  SET_CD_PARAMS (0)
  TRIGGER WHEN DISTANCE = 1 DELAY = ArcGetDelay(#PreDefinition, WDAT1) DO ArcMainNG(#PreDefinition, WDAT1, WP3) PRIO = -1
  TRIGGER WHEN PATH = ArcGetPath(#OnTheFlyArcOn, WDAT1) DELAY = ArcGetDelay(#GasPreflow, WDAT1) DO ArcMainNG(#GasPreflow, WDAT1, WP3) PRIO = -1
  TRIGGER WHEN PATH = ArcGetPath(#OnTheFlyArcOn, WDAT1) DELAY = 0 DO ArcMainNG(#ArcOnMoveStd, WDAT1, WP3) PRIO = -1
  ArcMainNG(#ArcOnBeforeMoveStd, WDAT1, WP3)
  LIN XP3
  ArcMainNG(#ArcOnAfterMoveStd, WDAT1, WP3)
;ENDFOLD
   $VEL.CP = 0.025
   LIN  {X -9.800, Y 9.800, Z 18.900, A 0.000, B 0.000, C 0.000} C_DIS
   $VEL.CP = 0.060
   LIN  {X -9.800, Y -9.800, Z 18.900, A 0.000, B 0.000, C 0.000} C_DIS
   $VEL.CP = 0.060
   LIN  {X 9.800, Y -9.800, Z 18.900, A 0.000, B 0.000, C 0.000} C_DIS
   $VEL.CP = 0.060
   LIN  {X 9.800, Y 9.800, Z 18.900, A 0.000, B 0.000, C 0.000} C_DIS
   $VEL.CP = 0.060
   LIN  {X -9.800, Y 9.800, Z 18.900, A 0.000, B 0.000, C 0.000} C_DIS

;FOLD ARCOFF WDAT2 LIN P4 CPDAT2 Tool[1]:cmttorch Base[1]:vrashatel ;%{PE}
  ;FOLD Parameters ;%{h}
    ;Params IlfProvider=kukaroboter.arctech.arcofflin; Kuka.IsGlobalPoint=False; Kuka.PointName=P4; Kuka.BlendingEnabled=False; Kuka.MoveDataName=CPDAT2; Kuka.VelocityPath=0.01; Kuka.CurrentCDSetIndex=0; Kuka.MovementParameterFieldEnabled=True; ArcTech.WdatVarName=WDAT2; ArcTech.Basic=3.4.3.1264
  ;ENDFOLD
  $BWDSTART = FALSE
  LDAT_ACT = LCPDAT2
  FDAT_ACT = FP4
  BAS(#CP_PARAMS, gArcBasVelDefinition)
  SET_CD_PARAMS (0)
  TRIGGER WHEN PATH = ArcGetPath(#ArcOffBefore, WDAT2) DELAY = 0 DO ArcMainNG(#ArcOffBeforeOffStd, WDAT2, WP4) PRIO = -1
  TRIGGER WHEN PATH = ArcGetPath(#OnTheFlyArcOff, WDAT2) DELAY = 0 DO ArcMainNG(#ArcOffMoveStd, WDAT2, WP4) PRIO = -1
  ArcMainNG(#ArcOffBeforeMoveStd, WDAT2, WP4)
  LIN XP4
  ArcMainNG(#ArcOffAfterMoveStd, WDAT2, WP4)
;ENDFOLD
   $VEL.CP = 0.080
   LIN  {X -9.800, Y 9.600, Z 18.900, A 0.000, B 0.000, C 0.000} C_DIS
   $VEL.CP = 0.080
   LIN  {X -9.360, Y 9.360, Z 18.900, A 0.000, B 0.000, C 0.000} C_DIS
   $VEL.CP = 0.080
   LIN  {X -4.094, Y 4.605, Z 18.900, A 0.000, B 0.000, C 0.000} C_DIS
   $VEL.CP = 0.080
   LIN  {X -3.794, Y 4.605, Z 18.900, A 0.000, B 0.000, C 0.000} C_DIS

;FOLD ARCON WDAT1 LIN P3 Vel=0.5 m/s CPDAT1 Tool[1]:cmttorch Base[1]:vrashatel ;%{PE}
  ;FOLD Parameters ;%{h}
    ;Params IlfProvider=kukaroboter.arctech.arconlin; Kuka.IsGlobalPoint=False; Kuka.PointName=P3; Kuka.BlendingEnabled=False; Kuka.MoveDataName=CPDAT1; Kuka.VelocityPath=0.5; Kuka.CurrentCDSetIndex=0; Kuka.MovementParameterFieldEnabled=True; ArcTech.WdatVarName=WDAT1; ArcTech.Basic=3.4.3.1264
  ;ENDFOLD
  $BWDSTART = FALSE
  LDAT_ACT = LCPDAT1
  FDAT_ACT = FP3
  BAS(#CP_PARAMS, 0.5)
  SET_CD_PARAMS (0)
  TRIGGER WHEN DISTANCE = 1 DELAY = ArcGetDelay(#PreDefinition, WDAT1) DO ArcMainNG(#PreDefinition, WDAT1, WP3) PRIO = -1
  TRIGGER WHEN PATH = ArcGetPath(#OnTheFlyArcOn, WDAT1) DELAY = ArcGetDelay(#GasPreflow, WDAT1) DO ArcMainNG(#GasPreflow, WDAT1, WP3) PRIO = -1
  TRIGGER WHEN PATH = ArcGetPath(#OnTheFlyArcOn, WDAT1) DELAY = 0 DO ArcMainNG(#ArcOnMoveStd, WDAT1, WP3) PRIO = -1
  ArcMainNG(#ArcOnBeforeMoveStd, WDAT1, WP3)
  LIN XP3
  ArcMainNG(#ArcOnAfterMoveStd, WDAT1, WP3)
;ENDFOLD
   $VEL.CP = 0.060
   LIN  {X -3.794, Y 6.518, Z 18.900, A 0.000, B 0.000, C 0.000} C_DIS
   $VEL.CP = 0.060
   LIN  {X 4.127, Y 6.518, Z 18.900, A 0.000, B 0.000, C 0.000} C_DIS
   $VEL.CP = 0.060
   LIN  {X 4.127, Y 5.850, Z 18.900, A 0.000, B 0.000, C 0.000} C_DIS
   $VEL.CP = 0.060
   LIN  {X -1.057, Y -4.280, Z 18.900, A 0.000, B 0.000, C 0.000} C_DIS
   $VEL.CP = 0.060
   LIN  {X 4.312, Y -4.280, Z 18.900, A 0.000, B 0.000, C 0.000} C_DIS
   $VEL.CP = 0.060
   LIN  {X 4.312, Y -6.193, Z 18.900, A 0.000, B 0.000, C 0.000} C_DIS
   $VEL.CP = 0.060
   LIN  {X -3.878, Y -6.193, Z 18.900, A 0.000, B 0.000, C 0.000} C_DIS
   $VEL.CP = 0.060
   LIN  {X -3.878, Y -5.525, Z 18.900, A 0.000, B 0.000, C 0.000} C_DIS
   $VEL.CP = 0.060
   LIN  {X 1.290, Y 4.605, Z 18.900, A 0.000, B 0.000, C 0.000} C_DIS
   $VEL.CP = 0.060
   LIN  {X -3.794, Y 4.605, Z 18.900, A 0.000, B 0.000, C 0.000} C_DIS

;FOLD ARCOFF WDAT2 LIN P4 CPDAT2 Tool[1]:cmttorch Base[1]:vrashatel ;%{PE}
  ;FOLD Parameters ;%{h}
    ;Params IlfProvider=kukaroboter.arctech.arcofflin; Kuka.IsGlobalPoint=False; Kuka.PointName=P4; Kuka.BlendingEnabled=False; Kuka.MoveDataName=CPDAT2; Kuka.VelocityPath=0.01; Kuka.CurrentCDSetIndex=0; Kuka.MovementParameterFieldEnabled=True; ArcTech.WdatVarName=WDAT2; ArcTech.Basic=3.4.3.1264
  ;ENDFOLD
  $BWDSTART = FALSE
  LDAT_ACT = LCPDAT2
  FDAT_ACT = FP4
  BAS(#CP_PARAMS, gArcBasVelDefinition)
  SET_CD_PARAMS (0)
  TRIGGER WHEN PATH = ArcGetPath(#ArcOffBefore, WDAT2) DELAY = 0 DO ArcMainNG(#ArcOffBeforeOffStd, WDAT2, WP4) PRIO = -1
  TRIGGER WHEN PATH = ArcGetPath(#OnTheFlyArcOff, WDAT2) DELAY = 0 DO ArcMainNG(#ArcOffMoveStd, WDAT2, WP4) PRIO = -1
  ArcMainNG(#ArcOffBeforeMoveStd, WDAT2, WP4)
  LIN XP4
  ArcMainNG(#ArcOffAfterMoveStd, WDAT2, WP4)
;ENDFOLD
   $VEL.CP = 0.080
   LIN  {X -3.794, Y 4.805, Z 18.900, A 0.000, B 0.000, C 0.000} C_DIS
   $VEL.CP = 0.080
   LIN  {X -4.194, Y 4.205, Z 18.900, A 0.000, B 0.000, C 0.000} C_DIS

;FOLD ARCON WDAT1 LIN P3 Vel=0.5 m/s CPDAT1 Tool[1]:cmttorch Base[1]:vrashatel ;%{PE}
  ;FOLD Parameters ;%{h}
    ;Params IlfProvider=kukaroboter.arctech.arconlin; Kuka.IsGlobalPoint=False; Kuka.PointName=P3; Kuka.BlendingEnabled=False; Kuka.MoveDataName=CPDAT1; Kuka.VelocityPath=0.5; Kuka.CurrentCDSetIndex=0; Kuka.MovementParameterFieldEnabled=True; ArcTech.WdatVarName=WDAT1; ArcTech.Basic=3.4.3.1264
  ;ENDFOLD
  $BWDSTART = FALSE
  LDAT_ACT = LCPDAT1
  FDAT_ACT = FP3
  BAS(#CP_PARAMS, 0.5)
  SET_CD_PARAMS (0)
  TRIGGER WHEN DISTANCE = 1 DELAY = ArcGetDelay(#PreDefinition, WDAT1) DO ArcMainNG(#PreDefinition, WDAT1, WP3) PRIO = -1
  TRIGGER WHEN PATH = ArcGetPath(#OnTheFlyArcOn, WDAT1) DELAY = ArcGetDelay(#GasPreflow, WDAT1) DO ArcMainNG(#GasPreflow, WDAT1, WP3) PRIO = -1
  TRIGGER WHEN PATH = ArcGetPath(#OnTheFlyArcOn, WDAT1) DELAY = 0 DO ArcMainNG(#ArcOnMoveStd, WDAT1, WP3) PRIO = -1
  ArcMainNG(#ArcOnBeforeMoveStd, WDAT1, WP3)
  LIN XP3
  ArcMainNG(#ArcOnAfterMoveStd, WDAT1, WP3)
;ENDFOLD
   $VEL.CP = 0.060
   LIN  {X -4.194, Y 6.918, Z 18.900, A 0.000, B 0.000, C 0.000} C_DIS
   $VEL.CP = 0.060
   LIN  {X 4.527, Y 6.918, Z 18.900, A 0.000, B 0.000, C 0.000} C_DIS
   $VEL.CP = 0.060
   LIN  {X 4.527, Y 5.754, Z 18.900, A 0.000, B 0.000, C 0.000} C_DIS
   $VEL.CP = 0.060
   LIN  {X -0.403, Y -3.880, Z 18.900, A 0.000, B 0.000, C 0.000} C_DIS
   $VEL.CP = 0.060
   LIN  {X 4.712, Y -3.880, Z 18.900, A 0.000, B 0.000, C 0.000} C_DIS
   $VEL.CP = 0.060
   LIN  {X 4.712, Y -6.593, Z 18.900, A 0.000, B 0.000, C 0.000} C_DIS
   $VEL.CP = 0.060
   LIN  {X -4.278, Y -6.593, Z 18.900, A 0.000, B 0.000, C 0.000} C_DIS
   $VEL.CP = 0.060
   LIN  {X -4.278, Y -5.429, Z 18.900, A 0.000, B 0.000, C 0.000} C_DIS
   $VEL.CP = 0.060
   LIN  {X 0.637, Y 4.205, Z 18.900, A 0.000, B 0.000, C 0.000} C_DIS
   $VEL.CP = 0.060
   LIN  {X -4.194, Y 4.205, Z 18.900, A 0.000, B 0.000, C 0.000} C_DIS

;FOLD ARCOFF WDAT2 LIN P4 CPDAT2 Tool[1]:cmttorch Base[1]:vrashatel ;%{PE}
  ;FOLD Parameters ;%{h}
    ;Params IlfProvider=kukaroboter.arctech.arcofflin; Kuka.IsGlobalPoint=False; Kuka.PointName=P4; Kuka.BlendingEnabled=False; Kuka.MoveDataName=CPDAT2; Kuka.VelocityPath=0.01; Kuka.CurrentCDSetIndex=0; Kuka.MovementParameterFieldEnabled=True; ArcTech.WdatVarName=WDAT2; ArcTech.Basic=3.4.3.1264
  ;ENDFOLD
  $BWDSTART = FALSE
  LDAT_ACT = LCPDAT2
  FDAT_ACT = FP4
  BAS(#CP_PARAMS, gArcBasVelDefinition)
  SET_CD_PARAMS (0)
  TRIGGER WHEN PATH = ArcGetPath(#ArcOffBefore, WDAT2) DELAY = 0 DO ArcMainNG(#ArcOffBeforeOffStd, WDAT2, WP4) PRIO = -1
  TRIGGER WHEN PATH = ArcGetPath(#OnTheFlyArcOff, WDAT2) DELAY = 0 DO ArcMainNG(#ArcOffMoveStd, WDAT2, WP4) PRIO = -1
  ArcMainNG(#ArcOffBeforeMoveStd, WDAT2, WP4)
  LIN XP4
  ArcMainNG(#ArcOffAfterMoveStd, WDAT2, WP4)
;ENDFOLD
   $VEL.CP = 0.080
   LIN  {X -9.400, Y 9.400, Z 18.900, A 0.000, B 0.000, C 0.000} C_DIS

;FOLD ARCON WDAT1 LIN P3 Vel=0.5 m/s CPDAT1 Tool[1]:cmttorch Base[1]:vrashatel ;%{PE}
  ;FOLD Parameters ;%{h}
    ;Params IlfProvider=kukaroboter.arctech.arconlin; Kuka.IsGlobalPoint=False; Kuka.PointName=P3; Kuka.BlendingEnabled=False; Kuka.MoveDataName=CPDAT1; Kuka.VelocityPath=0.5; Kuka.CurrentCDSetIndex=0; Kuka.MovementParameterFieldEnabled=True; ArcTech.WdatVarName=WDAT1; ArcTech.Basic=3.4.3.1264
  ;ENDFOLD
  $BWDSTART = FALSE
  LDAT_ACT = LCPDAT1
  FDAT_ACT = FP3
  BAS(#CP_PARAMS, 0.5)
  SET_CD_PARAMS (0)
  TRIGGER WHEN DISTANCE = 1 DELAY = ArcGetDelay(#PreDefinition, WDAT1) DO ArcMainNG(#PreDefinition, WDAT1, WP3) PRIO = -1
  TRIGGER WHEN PATH = ArcGetPath(#OnTheFlyArcOn, WDAT1) DELAY = ArcGetDelay(#GasPreflow, WDAT1) DO ArcMainNG(#GasPreflow, WDAT1, WP3) PRIO = -1
  TRIGGER WHEN PATH = ArcGetPath(#OnTheFlyArcOn, WDAT1) DELAY = 0 DO ArcMainNG(#ArcOnMoveStd, WDAT1, WP3) PRIO = -1
  ArcMainNG(#ArcOnBeforeMoveStd, WDAT1, WP3)
  LIN XP3
  ArcMainNG(#ArcOnAfterMoveStd, WDAT1, WP3)
;ENDFOLD
   $VEL.CP = 0.060
   LIN  {X -9.400, Y -9.400, Z 18.900, A 0.000, B 0.000, C 0.000} C_DIS
   $VEL.CP = 0.060
   LIN  {X 9.400, Y -9.400, Z 18.900, A 0.000, B 0.000, C 0.000} C_DIS
   $VEL.CP = 0.060
   LIN  {X 9.400, Y 9.400, Z 18.900, A 0.000, B 0.000, C 0.000} C_DIS
   $VEL.CP = 0.060
   LIN  {X -9.400, Y 9.400, Z 18.900, A 0.000, B 0.000, C 0.000} C_DIS

;FOLD ARCOFF WDAT2 LIN P4 CPDAT2 Tool[1]:cmttorch Base[1]:vrashatel ;%{PE}
  ;FOLD Parameters ;%{h}
    ;Params IlfProvider=kukaroboter.arctech.arcofflin; Kuka.IsGlobalPoint=False; Kuka.PointName=P4; Kuka.BlendingEnabled=False; Kuka.MoveDataName=CPDAT2; Kuka.VelocityPath=0.01; Kuka.CurrentCDSetIndex=0; Kuka.MovementParameterFieldEnabled=True; ArcTech.WdatVarName=WDAT2; ArcTech.Basic=3.4.3.1264
  ;ENDFOLD
  $BWDSTART = FALSE
  LDAT_ACT = LCPDAT2
  FDAT_ACT = FP4
  BAS(#CP_PARAMS, gArcBasVelDefinition)
  SET_CD_PARAMS (0)
  TRIGGER WHEN PATH = ArcGetPath(#ArcOffBefore, WDAT2) DELAY = 0 DO ArcMainNG(#ArcOffBeforeOffStd, WDAT2, WP4) PRIO = -1
  TRIGGER WHEN PATH = ArcGetPath(#OnTheFlyArcOff, WDAT2) DELAY = 0 DO ArcMainNG(#ArcOffMoveStd, WDAT2, WP4) PRIO = -1
  ArcMainNG(#ArcOffBeforeMoveStd, WDAT2, WP4)
  LIN XP4
  ArcMainNG(#ArcOffAfterMoveStd, WDAT2, WP4)
;ENDFOLD
   $VEL.CP = 0.080
   LIN  {X -9.040, Y 9.040, Z 18.900, A 0.000, B 0.000, C 0.000} C_DIS

;FOLD ARCON WDAT1 LIN P3 Vel=0.5 m/s CPDAT1 Tool[1]:cmttorch Base[1]:vrashatel ;%{PE}
  ;FOLD Parameters ;%{h}
    ;Params IlfProvider=kukaroboter.arctech.arconlin; Kuka.IsGlobalPoint=False; Kuka.PointName=P3; Kuka.BlendingEnabled=False; Kuka.MoveDataName=CPDAT1; Kuka.VelocityPath=0.5; Kuka.CurrentCDSetIndex=0; Kuka.MovementParameterFieldEnabled=True; ArcTech.WdatVarName=WDAT1; ArcTech.Basic=3.4.3.1264
  ;ENDFOLD
  $BWDSTART = FALSE
  LDAT_ACT = LCPDAT1
  FDAT_ACT = FP3
  BAS(#CP_PARAMS, 0.5)
  SET_CD_PARAMS (0)
  TRIGGER WHEN DISTANCE = 1 DELAY = ArcGetDelay(#PreDefinition, WDAT1) DO ArcMainNG(#PreDefinition, WDAT1, WP3) PRIO = -1
  TRIGGER WHEN PATH = ArcGetPath(#OnTheFlyArcOn, WDAT1) DELAY = ArcGetDelay(#GasPreflow, WDAT1) DO ArcMainNG(#GasPreflow, WDAT1, WP3) PRIO = -1
  TRIGGER WHEN PATH = ArcGetPath(#OnTheFlyArcOn, WDAT1) DELAY = 0 DO ArcMainNG(#ArcOnMoveStd, WDAT1, WP3) PRIO = -1
  ArcMainNG(#ArcOnBeforeMoveStd, WDAT1, WP3)
  LIN XP3
  ArcMainNG(#ArcOnAfterMoveStd, WDAT1, WP3)
;ENDFOLD
   $VEL.CP = 0.060
   LIN  {X -9.039, Y 5.102, Z 18.900, A 0.000, B 0.000, C 0.000} C_DIS
   $VEL.CP = 0.060
   LIN  {X -5.102, Y 9.039, Z 18.900, A 0.000, B 0.000, C 0.000} C_DIS
   $VEL.CP = 0.060
   LIN  {X -1.968, Y 9.039, Z 18.900, A 0.000, B 0.000, C 0.000} C_DIS
   $VEL.CP = 0.060
   LIN  {X -0.205, Y 7.276, Z 18.900, A 0.000, B 0.000, C 0.000} C_DIS
   $VEL.CP = 0.060
   LIN  {X 0.206, Y 7.277, Z 18.900, A 0.000, B 0.000, C 0.000} C_DIS
   $VEL.CP = 0.060
   LIN  {X 1.968, Y 9.039, Z 18.900, A 0.000, B 0.000, C 0.000} C_DIS
   $VEL.CP = 0.060
   LIN  {X 5.102, Y 9.039, Z 18.900, A 0.000, B 0.000, C 0.000} C_DIS
   $VEL.CP = 0.060
   LIN  {X 9.039, Y 5.102, Z 18.900, A 0.000, B 0.000, C 0.000} C_DIS
   $VEL.CP = 0.060
   LIN  {X 9.040, Y 9.040, Z 18.900, A 0.000, B 0.000, C 0.000} C_DIS
   $VEL.CP = 0.060
   LIN  {X 9.039, Y 9.039, Z 18.900, A 0.000, B 0.000, C 0.000} C_DIS
   $VEL.CP = 0.060
   LIN  {X 4.069, Y 4.069, Z 18.900, A 0.000, B 0.000, C 0.000} C_DIS
   $VEL.CP = 0.060
   LIN  {X 3.708, Y 3.362, Z 18.900, A 0.000, B 0.000, C 0.000} C_DIS
   $VEL.CP = 0.060
   LIN  {X 9.039, Y -1.968, Z 18.900, A 0.000, B 0.000, C 0.000} C_DIS
   $VEL.CP = 0.060
   LIN  {X 9.039, Y 1.968, Z 18.900, A 0.000, B 0.000, C 0.000} C_DIS
   $VEL.CP = 0.060
   LIN  {X 3.551, Y -3.519, Z 18.900, A 0.000, B 0.000, C 0.000} C_DIS
   $VEL.CP = 0.060
   LIN  {X 0.185, Y -3.520, Z 18.900, A 0.000, B 0.000, C 0.000} C_DIS
   $VEL.CP = 0.060
   LIN  {X 1.313, Y -1.313, Z 18.900, A 0.000, B 0.000, C 0.000} C_DIS
   $VEL.CP = 0.060
   LIN  {X 3.519, Y -3.519, Z 18.900, A 0.000, B 0.000, C 0.000} C_DIS

;FOLD ARCOFF WDAT2 LIN P4 CPDAT2 Tool[1]:cmttorch Base[1]:vrashatel ;%{PE}
  ;FOLD Parameters ;%{h}
    ;Params IlfProvider=kukaroboter.arctech.arcofflin; Kuka.IsGlobalPoint=False; Kuka.PointName=P4; Kuka.BlendingEnabled=False; Kuka.MoveDataName=CPDAT2; Kuka.VelocityPath=0.01; Kuka.CurrentCDSetIndex=0; Kuka.MovementParameterFieldEnabled=True; ArcTech.WdatVarName=WDAT2; ArcTech.Basic=3.4.3.1264
  ;ENDFOLD
  $BWDSTART = FALSE
  LDAT_ACT = LCPDAT2
  FDAT_ACT = FP4
  BAS(#CP_PARAMS, gArcBasVelDefinition)
  SET_CD_PARAMS (0)
  TRIGGER WHEN PATH = ArcGetPath(#ArcOffBefore, WDAT2) DELAY = 0 DO ArcMainNG(#ArcOffBeforeOffStd, WDAT2, WP4) PRIO = -1
  TRIGGER WHEN PATH = ArcGetPath(#OnTheFlyArcOff, WDAT2) DELAY = 0 DO ArcMainNG(#ArcOffMoveStd, WDAT2, WP4) PRIO = -1
  ArcMainNG(#ArcOffBeforeMoveStd, WDAT2, WP4)
  LIN XP4
  ArcMainNG(#ArcOffAfterMoveStd, WDAT2, WP4)
;ENDFOLD
   $VEL.CP = 0.060
   LIN  {X 3.589, Y -3.589, Z 18.900, A 0.000, B 0.000, C 0.000} C_DIS
   $VEL.CP = 0.080
   LIN  {X 4.540, Y -4.052, Z 18.900, A 0.000, B 0.000, C 0.000} C_DIS
   $VEL.CP = 0.080
   LIN  {X 5.072, Y -6.953, Z 18.900, A 0.000, B 0.000, C 0.000} C_DIS

;FOLD ARCON WDAT1 LIN P3 Vel=0.5 m/s CPDAT1 Tool[1]:cmttorch Base[1]:vrashatel ;%{PE}
  ;FOLD Parameters ;%{h}
    ;Params IlfProvider=kukaroboter.arctech.arconlin; Kuka.IsGlobalPoint=False; Kuka.PointName=P3; Kuka.BlendingEnabled=False; Kuka.MoveDataName=CPDAT1; Kuka.VelocityPath=0.5; Kuka.CurrentCDSetIndex=0; Kuka.MovementParameterFieldEnabled=True; ArcTech.WdatVarName=WDAT1; ArcTech.Basic=3.4.3.1264
  ;ENDFOLD
  $BWDSTART = FALSE
  LDAT_ACT = LCPDAT1
  FDAT_ACT = FP3
  BAS(#CP_PARAMS, 0.5)
  SET_CD_PARAMS (0)
  TRIGGER WHEN DISTANCE = 1 DELAY = ArcGetDelay(#PreDefinition, WDAT1) DO ArcMainNG(#PreDefinition, WDAT1, WP3) PRIO = -1
  TRIGGER WHEN PATH = ArcGetPath(#OnTheFlyArcOn, WDAT1) DELAY = ArcGetDelay(#GasPreflow, WDAT1) DO ArcMainNG(#GasPreflow, WDAT1, WP3) PRIO = -1
  TRIGGER WHEN PATH = ArcGetPath(#OnTheFlyArcOn, WDAT1) DELAY = 0 DO ArcMainNG(#ArcOnMoveStd, WDAT1, WP3) PRIO = -1
  ArcMainNG(#ArcOnBeforeMoveStd, WDAT1, WP3)
  LIN XP3
  ArcMainNG(#ArcOnAfterMoveStd, WDAT1, WP3)
;ENDFOLD
   $VEL.CP = 0.060
   LIN  {X 5.071, Y -5.071, Z 18.900, A 0.000, B 0.000, C 0.000} C_DIS
   $VEL.CP = 0.060
   LIN  {X 9.039, Y -9.039, Z 18.900, A 0.000, B 0.000, C 0.000} C_DIS
   $VEL.CP = 0.060
   LIN  {X 9.039, Y -5.102, Z 18.900, A 0.000, B 0.000, C 0.000} C_DIS
   $VEL.CP = 0.060
   LIN  {X 5.102, Y -9.039, Z 18.900, A 0.000, B 0.000, C 0.000} C_DIS
   $VEL.CP = 0.060
   LIN  {X 1.968, Y -9.039, Z 18.900, A 0.000, B 0.000, C 0.000} C_DIS
   $VEL.CP = 0.060
   LIN  {X -0.118, Y -6.952, Z 18.900, A 0.000, B 0.000, C 0.000} C_DIS
   $VEL.CP = 0.060
   LIN  {X 0.118, Y -6.952, Z 18.900, A 0.000, B 0.000, C 0.000} C_DIS
   $VEL.CP = 0.060
   LIN  {X -1.968, Y -9.039, Z 18.900, A 0.000, B 0.000, C 0.000} C_DIS
   $VEL.CP = 0.060
   LIN  {X -5.102, Y -9.039, Z 18.900, A 0.000, B 0.000, C 0.000} C_DIS
   $VEL.CP = 0.060
   LIN  {X -9.039, Y -5.102, Z 18.900, A 0.000, B 0.000, C 0.000} C_DIS
   $VEL.CP = 0.060
   LIN  {X -9.039, Y -9.039, Z 18.900, A 0.000, B 0.000, C 0.000} C_DIS
   $VEL.CP = 0.060
   LIN  {X -3.903, Y -3.903, Z 18.900, A 0.000, B 0.000, C 0.000} C_DIS
   $VEL.CP = 0.060
   LIN  {X -3.655, Y -3.415, Z 18.900, A 0.000, B 0.000, C 0.000} C_DIS
   $VEL.CP = 0.060
   LIN  {X -9.039, Y 1.968, Z 18.900, A 0.000, B 0.000, C 0.000} C_DIS
   $VEL.CP = 0.060
   LIN  {X -9.039, Y -1.968, Z 18.900, A 0.000, B 0.000, C 0.000} C_DIS
   $VEL.CP = 0.060
   LIN  {X -3.226, Y 3.844, Z 18.900, A 0.000, B 0.000, C 0.000} C_DIS
   $VEL.CP = 0.060
   LIN  {X 0.049, Y 3.845, Z 18.900, A 0.000, B 0.000, C 0.000} C_DIS
   $VEL.CP = 0.060
   LIN  {X -1.267, Y 1.267, Z 18.900, A 0.000, B 0.000, C 0.000} C_DIS
   $VEL.CP = 0.060
   LIN  {X -3.844, Y 3.844, Z 18.900, A 0.000, B 0.000, C 0.000} C_DIS
   $VEL.CP = 0.060
   LIN  {X -4.554, Y 3.845, Z 18.900, A 0.000, B 0.000, C 0.000} C_DIS
   $VEL.CP = 0.060
   LIN  {X -4.553, Y 4.553, Z 18.900, A 0.000, B 0.000, C 0.000} C_DIS
   $VEL.CP = 0.060
   LIN  {X -9.039, Y 9.039, Z 18.900, A 0.000, B 0.000, C 0.000} C_DIS
   $VEL.CP = 0.060
   LIN  {X -9.040, Y 9.040, Z 18.900, A 0.000, B 0.000, C 0.000} C_DIS

;FOLD ARCOFF WDAT2 LIN P4 CPDAT2 Tool[1]:cmttorch Base[1]:vrashatel ;%{PE}
  ;FOLD Parameters ;%{h}
    ;Params IlfProvider=kukaroboter.arctech.arcofflin; Kuka.IsGlobalPoint=False; Kuka.PointName=P4; Kuka.BlendingEnabled=False; Kuka.MoveDataName=CPDAT2; Kuka.VelocityPath=0.01; Kuka.CurrentCDSetIndex=0; Kuka.MovementParameterFieldEnabled=True; ArcTech.WdatVarName=WDAT2; ArcTech.Basic=3.4.3.1264
  ;ENDFOLD
  $BWDSTART = FALSE
  LDAT_ACT = LCPDAT2
  FDAT_ACT = FP4
  BAS(#CP_PARAMS, gArcBasVelDefinition)
  SET_CD_PARAMS (0)
  TRIGGER WHEN PATH = ArcGetPath(#ArcOffBefore, WDAT2) DELAY = 0 DO ArcMainNG(#ArcOffBeforeOffStd, WDAT2, WP4) PRIO = -1
  TRIGGER WHEN PATH = ArcGetPath(#OnTheFlyArcOff, WDAT2) DELAY = 0 DO ArcMainNG(#ArcOffMoveStd, WDAT2, WP4) PRIO = -1
  ArcMainNG(#ArcOffBeforeMoveStd, WDAT2, WP4)
  LIN XP4
  ArcMainNG(#ArcOffAfterMoveStd, WDAT2, WP4)
;ENDFOLD
   $VEL.CP = 0.010
   LIN  {X -9.040, Y 9.040, Z 19.100, A 0.000, B 0.000, C 0.000} C_DIS
   $VEL.CP = 0.080
   LIN  {X -9.530, Y 9.530, Z 19.100, A 0.000, B 0.000, C 0.000} C_DIS
   $VEL.CP = 0.080
   LIN  {X -9.800, Y 9.800, Z 19.100, A 0.000, B 0.000, C 0.000} C_DIS

;FOLD ARCON WDAT1 LIN P3 Vel=0.5 m/s CPDAT1 Tool[1]:cmttorch Base[1]:vrashatel ;%{PE}
  ;FOLD Parameters ;%{h}
    ;Params IlfProvider=kukaroboter.arctech.arconlin; Kuka.IsGlobalPoint=False; Kuka.PointName=P3; Kuka.BlendingEnabled=False; Kuka.MoveDataName=CPDAT1; Kuka.VelocityPath=0.5; Kuka.CurrentCDSetIndex=0; Kuka.MovementParameterFieldEnabled=True; ArcTech.WdatVarName=WDAT1; ArcTech.Basic=3.4.3.1264
  ;ENDFOLD
  $BWDSTART = FALSE
  LDAT_ACT = LCPDAT1
  FDAT_ACT = FP3
  BAS(#CP_PARAMS, 0.5)
  SET_CD_PARAMS (0)
  TRIGGER WHEN DISTANCE = 1 DELAY = ArcGetDelay(#PreDefinition, WDAT1) DO ArcMainNG(#PreDefinition, WDAT1, WP3) PRIO = -1
  TRIGGER WHEN PATH = ArcGetPath(#OnTheFlyArcOn, WDAT1) DELAY = ArcGetDelay(#GasPreflow, WDAT1) DO ArcMainNG(#GasPreflow, WDAT1, WP3) PRIO = -1
  TRIGGER WHEN PATH = ArcGetPath(#OnTheFlyArcOn, WDAT1) DELAY = 0 DO ArcMainNG(#ArcOnMoveStd, WDAT1, WP3) PRIO = -1
  ArcMainNG(#ArcOnBeforeMoveStd, WDAT1, WP3)
  LIN XP3
  ArcMainNG(#ArcOnAfterMoveStd, WDAT1, WP3)
;ENDFOLD
   $VEL.CP = 0.025
   LIN  {X -9.800, Y 9.800, Z 19.100, A 0.000, B 0.000, C 0.000} C_DIS
   $VEL.CP = 0.060
   LIN  {X -9.800, Y -9.800, Z 19.100, A 0.000, B 0.000, C 0.000} C_DIS
   $VEL.CP = 0.060
   LIN  {X 9.800, Y -9.800, Z 19.100, A 0.000, B 0.000, C 0.000} C_DIS
   $VEL.CP = 0.060
   LIN  {X 9.800, Y 9.800, Z 19.100, A 0.000, B 0.000, C 0.000} C_DIS
   $VEL.CP = 0.060
   LIN  {X -9.800, Y 9.800, Z 19.100, A 0.000, B 0.000, C 0.000} C_DIS

;FOLD ARCOFF WDAT2 LIN P4 CPDAT2 Tool[1]:cmttorch Base[1]:vrashatel ;%{PE}
  ;FOLD Parameters ;%{h}
    ;Params IlfProvider=kukaroboter.arctech.arcofflin; Kuka.IsGlobalPoint=False; Kuka.PointName=P4; Kuka.BlendingEnabled=False; Kuka.MoveDataName=CPDAT2; Kuka.VelocityPath=0.01; Kuka.CurrentCDSetIndex=0; Kuka.MovementParameterFieldEnabled=True; ArcTech.WdatVarName=WDAT2; ArcTech.Basic=3.4.3.1264
  ;ENDFOLD
  $BWDSTART = FALSE
  LDAT_ACT = LCPDAT2
  FDAT_ACT = FP4
  BAS(#CP_PARAMS, gArcBasVelDefinition)
  SET_CD_PARAMS (0)
  TRIGGER WHEN PATH = ArcGetPath(#ArcOffBefore, WDAT2) DELAY = 0 DO ArcMainNG(#ArcOffBeforeOffStd, WDAT2, WP4) PRIO = -1
  TRIGGER WHEN PATH = ArcGetPath(#OnTheFlyArcOff, WDAT2) DELAY = 0 DO ArcMainNG(#ArcOffMoveStd, WDAT2, WP4) PRIO = -1
  ArcMainNG(#ArcOffBeforeMoveStd, WDAT2, WP4)
  LIN XP4
  ArcMainNG(#ArcOffAfterMoveStd, WDAT2, WP4)
;ENDFOLD
   $VEL.CP = 0.080
   LIN  {X -9.800, Y 9.600, Z 19.100, A 0.000, B 0.000, C 0.000} C_DIS
   $VEL.CP = 0.080
   LIN  {X -9.360, Y 9.360, Z 19.100, A 0.000, B 0.000, C 0.000} C_DIS
   $VEL.CP = 0.080
   LIN  {X -4.094, Y 4.605, Z 19.100, A 0.000, B 0.000, C 0.000} C_DIS
   $VEL.CP = 0.080
   LIN  {X -3.794, Y 4.605, Z 19.100, A 0.000, B 0.000, C 0.000} C_DIS

;FOLD ARCON WDAT1 LIN P3 Vel=0.5 m/s CPDAT1 Tool[1]:cmttorch Base[1]:vrashatel ;%{PE}
  ;FOLD Parameters ;%{h}
    ;Params IlfProvider=kukaroboter.arctech.arconlin; Kuka.IsGlobalPoint=False; Kuka.PointName=P3; Kuka.BlendingEnabled=False; Kuka.MoveDataName=CPDAT1; Kuka.VelocityPath=0.5; Kuka.CurrentCDSetIndex=0; Kuka.MovementParameterFieldEnabled=True; ArcTech.WdatVarName=WDAT1; ArcTech.Basic=3.4.3.1264
  ;ENDFOLD
  $BWDSTART = FALSE
  LDAT_ACT = LCPDAT1
  FDAT_ACT = FP3
  BAS(#CP_PARAMS, 0.5)
  SET_CD_PARAMS (0)
  TRIGGER WHEN DISTANCE = 1 DELAY = ArcGetDelay(#PreDefinition, WDAT1) DO ArcMainNG(#PreDefinition, WDAT1, WP3) PRIO = -1
  TRIGGER WHEN PATH = ArcGetPath(#OnTheFlyArcOn, WDAT1) DELAY = ArcGetDelay(#GasPreflow, WDAT1) DO ArcMainNG(#GasPreflow, WDAT1, WP3) PRIO = -1
  TRIGGER WHEN PATH = ArcGetPath(#OnTheFlyArcOn, WDAT1) DELAY = 0 DO ArcMainNG(#ArcOnMoveStd, WDAT1, WP3) PRIO = -1
  ArcMainNG(#ArcOnBeforeMoveStd, WDAT1, WP3)
  LIN XP3
  ArcMainNG(#ArcOnAfterMoveStd, WDAT1, WP3)
;ENDFOLD
   $VEL.CP = 0.060
   LIN  {X -3.794, Y 6.518, Z 19.100, A 0.000, B 0.000, C 0.000} C_DIS
   $VEL.CP = 0.060
   LIN  {X 4.127, Y 6.518, Z 19.100, A 0.000, B 0.000, C 0.000} C_DIS
   $VEL.CP = 0.060
   LIN  {X 4.127, Y 5.850, Z 19.100, A 0.000, B 0.000, C 0.000} C_DIS
   $VEL.CP = 0.060
   LIN  {X -1.057, Y -4.280, Z 19.100, A 0.000, B 0.000, C 0.000} C_DIS
   $VEL.CP = 0.060
   LIN  {X 4.312, Y -4.280, Z 19.100, A 0.000, B 0.000, C 0.000} C_DIS
   $VEL.CP = 0.060
   LIN  {X 4.312, Y -6.193, Z 19.100, A 0.000, B 0.000, C 0.000} C_DIS
   $VEL.CP = 0.060
   LIN  {X -3.878, Y -6.193, Z 19.100, A 0.000, B 0.000, C 0.000} C_DIS
   $VEL.CP = 0.060
   LIN  {X -3.878, Y -5.525, Z 19.100, A 0.000, B 0.000, C 0.000} C_DIS
   $VEL.CP = 0.060
   LIN  {X 1.290, Y 4.605, Z 19.100, A 0.000, B 0.000, C 0.000} C_DIS
   $VEL.CP = 0.060
   LIN  {X -3.794, Y 4.605, Z 19.100, A 0.000, B 0.000, C 0.000} C_DIS

;FOLD ARCOFF WDAT2 LIN P4 CPDAT2 Tool[1]:cmttorch Base[1]:vrashatel ;%{PE}
  ;FOLD Parameters ;%{h}
    ;Params IlfProvider=kukaroboter.arctech.arcofflin; Kuka.IsGlobalPoint=False; Kuka.PointName=P4; Kuka.BlendingEnabled=False; Kuka.MoveDataName=CPDAT2; Kuka.VelocityPath=0.01; Kuka.CurrentCDSetIndex=0; Kuka.MovementParameterFieldEnabled=True; ArcTech.WdatVarName=WDAT2; ArcTech.Basic=3.4.3.1264
  ;ENDFOLD
  $BWDSTART = FALSE
  LDAT_ACT = LCPDAT2
  FDAT_ACT = FP4
  BAS(#CP_PARAMS, gArcBasVelDefinition)
  SET_CD_PARAMS (0)
  TRIGGER WHEN PATH = ArcGetPath(#ArcOffBefore, WDAT2) DELAY = 0 DO ArcMainNG(#ArcOffBeforeOffStd, WDAT2, WP4) PRIO = -1
  TRIGGER WHEN PATH = ArcGetPath(#OnTheFlyArcOff, WDAT2) DELAY = 0 DO ArcMainNG(#ArcOffMoveStd, WDAT2, WP4) PRIO = -1
  ArcMainNG(#ArcOffBeforeMoveStd, WDAT2, WP4)
  LIN XP4
  ArcMainNG(#ArcOffAfterMoveStd, WDAT2, WP4)
;ENDFOLD
   $VEL.CP = 0.080
   LIN  {X -3.794, Y 4.805, Z 19.100, A 0.000, B 0.000, C 0.000} C_DIS
   $VEL.CP = 0.080
   LIN  {X -4.194, Y 4.205, Z 19.100, A 0.000, B 0.000, C 0.000} C_DIS

;FOLD ARCON WDAT1 LIN P3 Vel=0.5 m/s CPDAT1 Tool[1]:cmttorch Base[1]:vrashatel ;%{PE}
  ;FOLD Parameters ;%{h}
    ;Params IlfProvider=kukaroboter.arctech.arconlin; Kuka.IsGlobalPoint=False; Kuka.PointName=P3; Kuka.BlendingEnabled=False; Kuka.MoveDataName=CPDAT1; Kuka.VelocityPath=0.5; Kuka.CurrentCDSetIndex=0; Kuka.MovementParameterFieldEnabled=True; ArcTech.WdatVarName=WDAT1; ArcTech.Basic=3.4.3.1264
  ;ENDFOLD
  $BWDSTART = FALSE
  LDAT_ACT = LCPDAT1
  FDAT_ACT = FP3
  BAS(#CP_PARAMS, 0.5)
  SET_CD_PARAMS (0)
  TRIGGER WHEN DISTANCE = 1 DELAY = ArcGetDelay(#PreDefinition, WDAT1) DO ArcMainNG(#PreDefinition, WDAT1, WP3) PRIO = -1
  TRIGGER WHEN PATH = ArcGetPath(#OnTheFlyArcOn, WDAT1) DELAY = ArcGetDelay(#GasPreflow, WDAT1) DO ArcMainNG(#GasPreflow, WDAT1, WP3) PRIO = -1
  TRIGGER WHEN PATH = ArcGetPath(#OnTheFlyArcOn, WDAT1) DELAY = 0 DO ArcMainNG(#ArcOnMoveStd, WDAT1, WP3) PRIO = -1
  ArcMainNG(#ArcOnBeforeMoveStd, WDAT1, WP3)
  LIN XP3
  ArcMainNG(#ArcOnAfterMoveStd, WDAT1, WP3)
;ENDFOLD
   $VEL.CP = 0.060
   LIN  {X -4.194, Y 6.918, Z 19.100, A 0.000, B 0.000, C 0.000} C_DIS
   $VEL.CP = 0.060
   LIN  {X 4.527, Y 6.918, Z 19.100, A 0.000, B 0.000, C 0.000} C_DIS
   $VEL.CP = 0.060
   LIN  {X 4.527, Y 5.754, Z 19.100, A 0.000, B 0.000, C 0.000} C_DIS
   $VEL.CP = 0.060
   LIN  {X -0.403, Y -3.880, Z 19.100, A 0.000, B 0.000, C 0.000} C_DIS
   $VEL.CP = 0.060
   LIN  {X 4.712, Y -3.880, Z 19.100, A 0.000, B 0.000, C 0.000} C_DIS
   $VEL.CP = 0.060
   LIN  {X 4.712, Y -6.593, Z 19.100, A 0.000, B 0.000, C 0.000} C_DIS
   $VEL.CP = 0.060
   LIN  {X -4.278, Y -6.593, Z 19.100, A 0.000, B 0.000, C 0.000} C_DIS
   $VEL.CP = 0.060
   LIN  {X -4.278, Y -5.429, Z 19.100, A 0.000, B 0.000, C 0.000} C_DIS
   $VEL.CP = 0.060
   LIN  {X 0.637, Y 4.205, Z 19.100, A 0.000, B 0.000, C 0.000} C_DIS
   $VEL.CP = 0.060
   LIN  {X -4.194, Y 4.205, Z 19.100, A 0.000, B 0.000, C 0.000} C_DIS

;FOLD ARCOFF WDAT2 LIN P4 CPDAT2 Tool[1]:cmttorch Base[1]:vrashatel ;%{PE}
  ;FOLD Parameters ;%{h}
    ;Params IlfProvider=kukaroboter.arctech.arcofflin; Kuka.IsGlobalPoint=False; Kuka.PointName=P4; Kuka.BlendingEnabled=False; Kuka.MoveDataName=CPDAT2; Kuka.VelocityPath=0.01; Kuka.CurrentCDSetIndex=0; Kuka.MovementParameterFieldEnabled=True; ArcTech.WdatVarName=WDAT2; ArcTech.Basic=3.4.3.1264
  ;ENDFOLD
  $BWDSTART = FALSE
  LDAT_ACT = LCPDAT2
  FDAT_ACT = FP4
  BAS(#CP_PARAMS, gArcBasVelDefinition)
  SET_CD_PARAMS (0)
  TRIGGER WHEN PATH = ArcGetPath(#ArcOffBefore, WDAT2) DELAY = 0 DO ArcMainNG(#ArcOffBeforeOffStd, WDAT2, WP4) PRIO = -1
  TRIGGER WHEN PATH = ArcGetPath(#OnTheFlyArcOff, WDAT2) DELAY = 0 DO ArcMainNG(#ArcOffMoveStd, WDAT2, WP4) PRIO = -1
  ArcMainNG(#ArcOffBeforeMoveStd, WDAT2, WP4)
  LIN XP4
  ArcMainNG(#ArcOffAfterMoveStd, WDAT2, WP4)
;ENDFOLD
   $VEL.CP = 0.080
   LIN  {X -9.400, Y 9.400, Z 19.100, A 0.000, B 0.000, C 0.000} C_DIS

;FOLD ARCON WDAT1 LIN P3 Vel=0.5 m/s CPDAT1 Tool[1]:cmttorch Base[1]:vrashatel ;%{PE}
  ;FOLD Parameters ;%{h}
    ;Params IlfProvider=kukaroboter.arctech.arconlin; Kuka.IsGlobalPoint=False; Kuka.PointName=P3; Kuka.BlendingEnabled=False; Kuka.MoveDataName=CPDAT1; Kuka.VelocityPath=0.5; Kuka.CurrentCDSetIndex=0; Kuka.MovementParameterFieldEnabled=True; ArcTech.WdatVarName=WDAT1; ArcTech.Basic=3.4.3.1264
  ;ENDFOLD
  $BWDSTART = FALSE
  LDAT_ACT = LCPDAT1
  FDAT_ACT = FP3
  BAS(#CP_PARAMS, 0.5)
  SET_CD_PARAMS (0)
  TRIGGER WHEN DISTANCE = 1 DELAY = ArcGetDelay(#PreDefinition, WDAT1) DO ArcMainNG(#PreDefinition, WDAT1, WP3) PRIO = -1
  TRIGGER WHEN PATH = ArcGetPath(#OnTheFlyArcOn, WDAT1) DELAY = ArcGetDelay(#GasPreflow, WDAT1) DO ArcMainNG(#GasPreflow, WDAT1, WP3) PRIO = -1
  TRIGGER WHEN PATH = ArcGetPath(#OnTheFlyArcOn, WDAT1) DELAY = 0 DO ArcMainNG(#ArcOnMoveStd, WDAT1, WP3) PRIO = -1
  ArcMainNG(#ArcOnBeforeMoveStd, WDAT1, WP3)
  LIN XP3
  ArcMainNG(#ArcOnAfterMoveStd, WDAT1, WP3)
;ENDFOLD
   $VEL.CP = 0.060
   LIN  {X -9.400, Y -9.400, Z 19.100, A 0.000, B 0.000, C 0.000} C_DIS
   $VEL.CP = 0.060
   LIN  {X 9.400, Y -9.400, Z 19.100, A 0.000, B 0.000, C 0.000} C_DIS
   $VEL.CP = 0.060
   LIN  {X 9.400, Y 9.400, Z 19.100, A 0.000, B 0.000, C 0.000} C_DIS
   $VEL.CP = 0.060
   LIN  {X -9.400, Y 9.400, Z 19.100, A 0.000, B 0.000, C 0.000} C_DIS

;FOLD ARCOFF WDAT2 LIN P4 CPDAT2 Tool[1]:cmttorch Base[1]:vrashatel ;%{PE}
  ;FOLD Parameters ;%{h}
    ;Params IlfProvider=kukaroboter.arctech.arcofflin; Kuka.IsGlobalPoint=False; Kuka.PointName=P4; Kuka.BlendingEnabled=False; Kuka.MoveDataName=CPDAT2; Kuka.VelocityPath=0.01; Kuka.CurrentCDSetIndex=0; Kuka.MovementParameterFieldEnabled=True; ArcTech.WdatVarName=WDAT2; ArcTech.Basic=3.4.3.1264
  ;ENDFOLD
  $BWDSTART = FALSE
  LDAT_ACT = LCPDAT2
  FDAT_ACT = FP4
  BAS(#CP_PARAMS, gArcBasVelDefinition)
  SET_CD_PARAMS (0)
  TRIGGER WHEN PATH = ArcGetPath(#ArcOffBefore, WDAT2) DELAY = 0 DO ArcMainNG(#ArcOffBeforeOffStd, WDAT2, WP4) PRIO = -1
  TRIGGER WHEN PATH = ArcGetPath(#OnTheFlyArcOff, WDAT2) DELAY = 0 DO ArcMainNG(#ArcOffMoveStd, WDAT2, WP4) PRIO = -1
  ArcMainNG(#ArcOffBeforeMoveStd, WDAT2, WP4)
  LIN XP4
  ArcMainNG(#ArcOffAfterMoveStd, WDAT2, WP4)
;ENDFOLD
   $VEL.CP = 0.080
   LIN  {X -9.040, Y 9.040, Z 19.100, A 0.000, B 0.000, C 0.000} C_DIS

;FOLD ARCON WDAT1 LIN P3 Vel=0.5 m/s CPDAT1 Tool[1]:cmttorch Base[1]:vrashatel ;%{PE}
  ;FOLD Parameters ;%{h}
    ;Params IlfProvider=kukaroboter.arctech.arconlin; Kuka.IsGlobalPoint=False; Kuka.PointName=P3; Kuka.BlendingEnabled=False; Kuka.MoveDataName=CPDAT1; Kuka.VelocityPath=0.5; Kuka.CurrentCDSetIndex=0; Kuka.MovementParameterFieldEnabled=True; ArcTech.WdatVarName=WDAT1; ArcTech.Basic=3.4.3.1264
  ;ENDFOLD
  $BWDSTART = FALSE
  LDAT_ACT = LCPDAT1
  FDAT_ACT = FP3
  BAS(#CP_PARAMS, 0.5)
  SET_CD_PARAMS (0)
  TRIGGER WHEN DISTANCE = 1 DELAY = ArcGetDelay(#PreDefinition, WDAT1) DO ArcMainNG(#PreDefinition, WDAT1, WP3) PRIO = -1
  TRIGGER WHEN PATH = ArcGetPath(#OnTheFlyArcOn, WDAT1) DELAY = ArcGetDelay(#GasPreflow, WDAT1) DO ArcMainNG(#GasPreflow, WDAT1, WP3) PRIO = -1
  TRIGGER WHEN PATH = ArcGetPath(#OnTheFlyArcOn, WDAT1) DELAY = 0 DO ArcMainNG(#ArcOnMoveStd, WDAT1, WP3) PRIO = -1
  ArcMainNG(#ArcOnBeforeMoveStd, WDAT1, WP3)
  LIN XP3
  ArcMainNG(#ArcOnAfterMoveStd, WDAT1, WP3)
;ENDFOLD
   $VEL.CP = 0.060
   LIN  {X -9.039, Y 5.102, Z 19.100, A 0.000, B 0.000, C 0.000} C_DIS
   $VEL.CP = 0.060
   LIN  {X -5.102, Y 9.039, Z 19.100, A 0.000, B 0.000, C 0.000} C_DIS
   $VEL.CP = 0.060
   LIN  {X -1.968, Y 9.039, Z 19.100, A 0.000, B 0.000, C 0.000} C_DIS
   $VEL.CP = 0.060
   LIN  {X -0.205, Y 7.276, Z 19.100, A 0.000, B 0.000, C 0.000} C_DIS
   $VEL.CP = 0.060
   LIN  {X 0.206, Y 7.277, Z 19.100, A 0.000, B 0.000, C 0.000} C_DIS
   $VEL.CP = 0.060
   LIN  {X 1.968, Y 9.039, Z 19.100, A 0.000, B 0.000, C 0.000} C_DIS
   $VEL.CP = 0.060
   LIN  {X 5.102, Y 9.039, Z 19.100, A 0.000, B 0.000, C 0.000} C_DIS
   $VEL.CP = 0.060
   LIN  {X 9.039, Y 5.102, Z 19.100, A 0.000, B 0.000, C 0.000} C_DIS
   $VEL.CP = 0.060
   LIN  {X 9.040, Y 9.040, Z 19.100, A 0.000, B 0.000, C 0.000} C_DIS
   $VEL.CP = 0.060
   LIN  {X 9.039, Y 9.039, Z 19.100, A 0.000, B 0.000, C 0.000} C_DIS
   $VEL.CP = 0.060
   LIN  {X 4.069, Y 4.069, Z 19.100, A 0.000, B 0.000, C 0.000} C_DIS
   $VEL.CP = 0.060
   LIN  {X 3.708, Y 3.362, Z 19.100, A 0.000, B 0.000, C 0.000} C_DIS
   $VEL.CP = 0.060
   LIN  {X 9.039, Y -1.968, Z 19.100, A 0.000, B 0.000, C 0.000} C_DIS
   $VEL.CP = 0.060
   LIN  {X 9.039, Y 1.968, Z 19.100, A 0.000, B 0.000, C 0.000} C_DIS
   $VEL.CP = 0.060
   LIN  {X 3.551, Y -3.519, Z 19.100, A 0.000, B 0.000, C 0.000} C_DIS
   $VEL.CP = 0.060
   LIN  {X 0.185, Y -3.520, Z 19.100, A 0.000, B 0.000, C 0.000} C_DIS
   $VEL.CP = 0.060
   LIN  {X 1.313, Y -1.313, Z 19.100, A 0.000, B 0.000, C 0.000} C_DIS
   $VEL.CP = 0.060
   LIN  {X 3.519, Y -3.519, Z 19.100, A 0.000, B 0.000, C 0.000} C_DIS

;FOLD ARCOFF WDAT2 LIN P4 CPDAT2 Tool[1]:cmttorch Base[1]:vrashatel ;%{PE}
  ;FOLD Parameters ;%{h}
    ;Params IlfProvider=kukaroboter.arctech.arcofflin; Kuka.IsGlobalPoint=False; Kuka.PointName=P4; Kuka.BlendingEnabled=False; Kuka.MoveDataName=CPDAT2; Kuka.VelocityPath=0.01; Kuka.CurrentCDSetIndex=0; Kuka.MovementParameterFieldEnabled=True; ArcTech.WdatVarName=WDAT2; ArcTech.Basic=3.4.3.1264
  ;ENDFOLD
  $BWDSTART = FALSE
  LDAT_ACT = LCPDAT2
  FDAT_ACT = FP4
  BAS(#CP_PARAMS, gArcBasVelDefinition)
  SET_CD_PARAMS (0)
  TRIGGER WHEN PATH = ArcGetPath(#ArcOffBefore, WDAT2) DELAY = 0 DO ArcMainNG(#ArcOffBeforeOffStd, WDAT2, WP4) PRIO = -1
  TRIGGER WHEN PATH = ArcGetPath(#OnTheFlyArcOff, WDAT2) DELAY = 0 DO ArcMainNG(#ArcOffMoveStd, WDAT2, WP4) PRIO = -1
  ArcMainNG(#ArcOffBeforeMoveStd, WDAT2, WP4)
  LIN XP4
  ArcMainNG(#ArcOffAfterMoveStd, WDAT2, WP4)
;ENDFOLD
   $VEL.CP = 0.060
   LIN  {X 3.589, Y -3.589, Z 19.100, A 0.000, B 0.000, C 0.000} C_DIS
   $VEL.CP = 0.080
   LIN  {X 4.540, Y -4.052, Z 19.100, A 0.000, B 0.000, C 0.000} C_DIS
   $VEL.CP = 0.080
   LIN  {X 5.072, Y -6.953, Z 19.100, A 0.000, B 0.000, C 0.000} C_DIS

;FOLD ARCON WDAT1 LIN P3 Vel=0.5 m/s CPDAT1 Tool[1]:cmttorch Base[1]:vrashatel ;%{PE}
  ;FOLD Parameters ;%{h}
    ;Params IlfProvider=kukaroboter.arctech.arconlin; Kuka.IsGlobalPoint=False; Kuka.PointName=P3; Kuka.BlendingEnabled=False; Kuka.MoveDataName=CPDAT1; Kuka.VelocityPath=0.5; Kuka.CurrentCDSetIndex=0; Kuka.MovementParameterFieldEnabled=True; ArcTech.WdatVarName=WDAT1; ArcTech.Basic=3.4.3.1264
  ;ENDFOLD
  $BWDSTART = FALSE
  LDAT_ACT = LCPDAT1
  FDAT_ACT = FP3
  BAS(#CP_PARAMS, 0.5)
  SET_CD_PARAMS (0)
  TRIGGER WHEN DISTANCE = 1 DELAY = ArcGetDelay(#PreDefinition, WDAT1) DO ArcMainNG(#PreDefinition, WDAT1, WP3) PRIO = -1
  TRIGGER WHEN PATH = ArcGetPath(#OnTheFlyArcOn, WDAT1) DELAY = ArcGetDelay(#GasPreflow, WDAT1) DO ArcMainNG(#GasPreflow, WDAT1, WP3) PRIO = -1
  TRIGGER WHEN PATH = ArcGetPath(#OnTheFlyArcOn, WDAT1) DELAY = 0 DO ArcMainNG(#ArcOnMoveStd, WDAT1, WP3) PRIO = -1
  ArcMainNG(#ArcOnBeforeMoveStd, WDAT1, WP3)
  LIN XP3
  ArcMainNG(#ArcOnAfterMoveStd, WDAT1, WP3)
;ENDFOLD
   $VEL.CP = 0.060
   LIN  {X 5.071, Y -5.071, Z 19.100, A 0.000, B 0.000, C 0.000} C_DIS
   $VEL.CP = 0.060
   LIN  {X 9.039, Y -9.039, Z 19.100, A 0.000, B 0.000, C 0.000} C_DIS
   $VEL.CP = 0.060
   LIN  {X 9.039, Y -5.102, Z 19.100, A 0.000, B 0.000, C 0.000} C_DIS
   $VEL.CP = 0.060
   LIN  {X 5.102, Y -9.039, Z 19.100, A 0.000, B 0.000, C 0.000} C_DIS
   $VEL.CP = 0.060
   LIN  {X 1.968, Y -9.039, Z 19.100, A 0.000, B 0.000, C 0.000} C_DIS
   $VEL.CP = 0.060
   LIN  {X -0.118, Y -6.952, Z 19.100, A 0.000, B 0.000, C 0.000} C_DIS
   $VEL.CP = 0.060
   LIN  {X 0.118, Y -6.952, Z 19.100, A 0.000, B 0.000, C 0.000} C_DIS
   $VEL.CP = 0.060
   LIN  {X -1.968, Y -9.039, Z 19.100, A 0.000, B 0.000, C 0.000} C_DIS
   $VEL.CP = 0.060
   LIN  {X -5.102, Y -9.039, Z 19.100, A 0.000, B 0.000, C 0.000} C_DIS
   $VEL.CP = 0.060
   LIN  {X -9.039, Y -5.102, Z 19.100, A 0.000, B 0.000, C 0.000} C_DIS
   $VEL.CP = 0.060
   LIN  {X -9.039, Y -9.039, Z 19.100, A 0.000, B 0.000, C 0.000} C_DIS
   $VEL.CP = 0.060
   LIN  {X -3.903, Y -3.903, Z 19.100, A 0.000, B 0.000, C 0.000} C_DIS
   $VEL.CP = 0.060
   LIN  {X -3.655, Y -3.415, Z 19.100, A 0.000, B 0.000, C 0.000} C_DIS
   $VEL.CP = 0.060
   LIN  {X -9.039, Y 1.968, Z 19.100, A 0.000, B 0.000, C 0.000} C_DIS
   $VEL.CP = 0.060
   LIN  {X -9.039, Y -1.968, Z 19.100, A 0.000, B 0.000, C 0.000} C_DIS
   $VEL.CP = 0.060
   LIN  {X -3.226, Y 3.844, Z 19.100, A 0.000, B 0.000, C 0.000} C_DIS
   $VEL.CP = 0.060
   LIN  {X 0.049, Y 3.845, Z 19.100, A 0.000, B 0.000, C 0.000} C_DIS
   $VEL.CP = 0.060
   LIN  {X -1.267, Y 1.267, Z 19.100, A 0.000, B 0.000, C 0.000} C_DIS
   $VEL.CP = 0.060
   LIN  {X -3.844, Y 3.844, Z 19.100, A 0.000, B 0.000, C 0.000} C_DIS
   $VEL.CP = 0.060
   LIN  {X -4.554, Y 3.845, Z 19.100, A 0.000, B 0.000, C 0.000} C_DIS
   $VEL.CP = 0.060
   LIN  {X -4.553, Y 4.553, Z 19.100, A 0.000, B 0.000, C 0.000} C_DIS
   $VEL.CP = 0.060
   LIN  {X -9.039, Y 9.039, Z 19.100, A 0.000, B 0.000, C 0.000} C_DIS
   $VEL.CP = 0.060
   LIN  {X -9.040, Y 9.040, Z 19.100, A 0.000, B 0.000, C 0.000} C_DIS

;FOLD ARCOFF WDAT2 LIN P4 CPDAT2 Tool[1]:cmttorch Base[1]:vrashatel ;%{PE}
  ;FOLD Parameters ;%{h}
    ;Params IlfProvider=kukaroboter.arctech.arcofflin; Kuka.IsGlobalPoint=False; Kuka.PointName=P4; Kuka.BlendingEnabled=False; Kuka.MoveDataName=CPDAT2; Kuka.VelocityPath=0.01; Kuka.CurrentCDSetIndex=0; Kuka.MovementParameterFieldEnabled=True; ArcTech.WdatVarName=WDAT2; ArcTech.Basic=3.4.3.1264
  ;ENDFOLD
  $BWDSTART = FALSE
  LDAT_ACT = LCPDAT2
  FDAT_ACT = FP4
  BAS(#CP_PARAMS, gArcBasVelDefinition)
  SET_CD_PARAMS (0)
  TRIGGER WHEN PATH = ArcGetPath(#ArcOffBefore, WDAT2) DELAY = 0 DO ArcMainNG(#ArcOffBeforeOffStd, WDAT2, WP4) PRIO = -1
  TRIGGER WHEN PATH = ArcGetPath(#OnTheFlyArcOff, WDAT2) DELAY = 0 DO ArcMainNG(#ArcOffMoveStd, WDAT2, WP4) PRIO = -1
  ArcMainNG(#ArcOffBeforeMoveStd, WDAT2, WP4)
  LIN XP4
  ArcMainNG(#ArcOffAfterMoveStd, WDAT2, WP4)
;ENDFOLD
   $VEL.CP = 0.010
   LIN  {X -9.040, Y 9.040, Z 19.300, A 0.000, B 0.000, C 0.000} C_DIS
   $VEL.CP = 0.080
   LIN  {X -9.530, Y 9.530, Z 19.300, A 0.000, B 0.000, C 0.000} C_DIS
   $VEL.CP = 0.080
   LIN  {X -9.800, Y 9.800, Z 19.300, A 0.000, B 0.000, C 0.000} C_DIS

;FOLD ARCON WDAT1 LIN P3 Vel=0.5 m/s CPDAT1 Tool[1]:cmttorch Base[1]:vrashatel ;%{PE}
  ;FOLD Parameters ;%{h}
    ;Params IlfProvider=kukaroboter.arctech.arconlin; Kuka.IsGlobalPoint=False; Kuka.PointName=P3; Kuka.BlendingEnabled=False; Kuka.MoveDataName=CPDAT1; Kuka.VelocityPath=0.5; Kuka.CurrentCDSetIndex=0; Kuka.MovementParameterFieldEnabled=True; ArcTech.WdatVarName=WDAT1; ArcTech.Basic=3.4.3.1264
  ;ENDFOLD
  $BWDSTART = FALSE
  LDAT_ACT = LCPDAT1
  FDAT_ACT = FP3
  BAS(#CP_PARAMS, 0.5)
  SET_CD_PARAMS (0)
  TRIGGER WHEN DISTANCE = 1 DELAY = ArcGetDelay(#PreDefinition, WDAT1) DO ArcMainNG(#PreDefinition, WDAT1, WP3) PRIO = -1
  TRIGGER WHEN PATH = ArcGetPath(#OnTheFlyArcOn, WDAT1) DELAY = ArcGetDelay(#GasPreflow, WDAT1) DO ArcMainNG(#GasPreflow, WDAT1, WP3) PRIO = -1
  TRIGGER WHEN PATH = ArcGetPath(#OnTheFlyArcOn, WDAT1) DELAY = 0 DO ArcMainNG(#ArcOnMoveStd, WDAT1, WP3) PRIO = -1
  ArcMainNG(#ArcOnBeforeMoveStd, WDAT1, WP3)
  LIN XP3
  ArcMainNG(#ArcOnAfterMoveStd, WDAT1, WP3)
;ENDFOLD
   $VEL.CP = 0.025
   LIN  {X -9.800, Y 9.800, Z 19.300, A 0.000, B 0.000, C 0.000} C_DIS
   $VEL.CP = 0.060
   LIN  {X -9.800, Y -9.800, Z 19.300, A 0.000, B 0.000, C 0.000} C_DIS
   $VEL.CP = 0.060
   LIN  {X 9.800, Y -9.800, Z 19.300, A 0.000, B 0.000, C 0.000} C_DIS
   $VEL.CP = 0.060
   LIN  {X 9.800, Y 9.800, Z 19.300, A 0.000, B 0.000, C 0.000} C_DIS
   $VEL.CP = 0.060
   LIN  {X -9.800, Y 9.800, Z 19.300, A 0.000, B 0.000, C 0.000} C_DIS

;FOLD ARCOFF WDAT2 LIN P4 CPDAT2 Tool[1]:cmttorch Base[1]:vrashatel ;%{PE}
  ;FOLD Parameters ;%{h}
    ;Params IlfProvider=kukaroboter.arctech.arcofflin; Kuka.IsGlobalPoint=False; Kuka.PointName=P4; Kuka.BlendingEnabled=False; Kuka.MoveDataName=CPDAT2; Kuka.VelocityPath=0.01; Kuka.CurrentCDSetIndex=0; Kuka.MovementParameterFieldEnabled=True; ArcTech.WdatVarName=WDAT2; ArcTech.Basic=3.4.3.1264
  ;ENDFOLD
  $BWDSTART = FALSE
  LDAT_ACT = LCPDAT2
  FDAT_ACT = FP4
  BAS(#CP_PARAMS, gArcBasVelDefinition)
  SET_CD_PARAMS (0)
  TRIGGER WHEN PATH = ArcGetPath(#ArcOffBefore, WDAT2) DELAY = 0 DO ArcMainNG(#ArcOffBeforeOffStd, WDAT2, WP4) PRIO = -1
  TRIGGER WHEN PATH = ArcGetPath(#OnTheFlyArcOff, WDAT2) DELAY = 0 DO ArcMainNG(#ArcOffMoveStd, WDAT2, WP4) PRIO = -1
  ArcMainNG(#ArcOffBeforeMoveStd, WDAT2, WP4)
  LIN XP4
  ArcMainNG(#ArcOffAfterMoveStd, WDAT2, WP4)
;ENDFOLD
   $VEL.CP = 0.080
   LIN  {X -9.800, Y 9.600, Z 19.300, A 0.000, B 0.000, C 0.000} C_DIS
   $VEL.CP = 0.080
   LIN  {X -9.360, Y 9.360, Z 19.300, A 0.000, B 0.000, C 0.000} C_DIS
   $VEL.CP = 0.080
   LIN  {X -4.094, Y 9.190, Z 19.300, A 0.000, B 0.000, C 0.000} C_DIS
   $VEL.CP = 0.080
   LIN  {X -4.094, Y 7.108, Z 19.300, A 0.000, B 0.000, C 0.000} C_DIS
   $VEL.CP = 0.080
   LIN  {X -4.094, Y 4.605, Z 19.300, A 0.000, B 0.000, C 0.000} C_DIS
   $VEL.CP = 0.080
   LIN  {X -3.794, Y 4.605, Z 19.300, A 0.000, B 0.000, C 0.000} C_DIS

;FOLD ARCON WDAT1 LIN P3 Vel=0.5 m/s CPDAT1 Tool[1]:cmttorch Base[1]:vrashatel ;%{PE}
  ;FOLD Parameters ;%{h}
    ;Params IlfProvider=kukaroboter.arctech.arconlin; Kuka.IsGlobalPoint=False; Kuka.PointName=P3; Kuka.BlendingEnabled=False; Kuka.MoveDataName=CPDAT1; Kuka.VelocityPath=0.5; Kuka.CurrentCDSetIndex=0; Kuka.MovementParameterFieldEnabled=True; ArcTech.WdatVarName=WDAT1; ArcTech.Basic=3.4.3.1264
  ;ENDFOLD
  $BWDSTART = FALSE
  LDAT_ACT = LCPDAT1
  FDAT_ACT = FP3
  BAS(#CP_PARAMS, 0.5)
  SET_CD_PARAMS (0)
  TRIGGER WHEN DISTANCE = 1 DELAY = ArcGetDelay(#PreDefinition, WDAT1) DO ArcMainNG(#PreDefinition, WDAT1, WP3) PRIO = -1
  TRIGGER WHEN PATH = ArcGetPath(#OnTheFlyArcOn, WDAT1) DELAY = ArcGetDelay(#GasPreflow, WDAT1) DO ArcMainNG(#GasPreflow, WDAT1, WP3) PRIO = -1
  TRIGGER WHEN PATH = ArcGetPath(#OnTheFlyArcOn, WDAT1) DELAY = 0 DO ArcMainNG(#ArcOnMoveStd, WDAT1, WP3) PRIO = -1
  ArcMainNG(#ArcOnBeforeMoveStd, WDAT1, WP3)
  LIN XP3
  ArcMainNG(#ArcOnAfterMoveStd, WDAT1, WP3)
;ENDFOLD
   $VEL.CP = 0.025
   LIN  {X -3.794, Y 4.605, Z 19.300, A 0.000, B 0.000, C 0.000} C_DIS
   $VEL.CP = 0.060
   LIN  {X -3.794, Y 6.518, Z 19.300, A 0.000, B 0.000, C 0.000} C_DIS
   $VEL.CP = 0.060
   LIN  {X 4.127, Y 6.518, Z 19.300, A 0.000, B 0.000, C 0.000} C_DIS
   $VEL.CP = 0.060
   LIN  {X 4.127, Y 5.850, Z 19.300, A 0.000, B 0.000, C 0.000} C_DIS
   $VEL.CP = 0.060
   LIN  {X -1.057, Y -4.280, Z 19.300, A 0.000, B 0.000, C 0.000} C_DIS
   $VEL.CP = 0.060
   LIN  {X 4.312, Y -4.280, Z 19.300, A 0.000, B 0.000, C 0.000} C_DIS
   $VEL.CP = 0.060
   LIN  {X 4.312, Y -6.193, Z 19.300, A 0.000, B 0.000, C 0.000} C_DIS
   $VEL.CP = 0.060
   LIN  {X -3.878, Y -6.193, Z 19.300, A 0.000, B 0.000, C 0.000} C_DIS
   $VEL.CP = 0.060
   LIN  {X -3.878, Y -5.525, Z 19.300, A 0.000, B 0.000, C 0.000} C_DIS
   $VEL.CP = 0.060
   LIN  {X 1.290, Y 4.605, Z 19.300, A 0.000, B 0.000, C 0.000} C_DIS
   $VEL.CP = 0.060
   LIN  {X -3.794, Y 4.605, Z 19.300, A 0.000, B 0.000, C 0.000} C_DIS

;FOLD ARCOFF WDAT2 LIN P4 CPDAT2 Tool[1]:cmttorch Base[1]:vrashatel ;%{PE}
  ;FOLD Parameters ;%{h}
    ;Params IlfProvider=kukaroboter.arctech.arcofflin; Kuka.IsGlobalPoint=False; Kuka.PointName=P4; Kuka.BlendingEnabled=False; Kuka.MoveDataName=CPDAT2; Kuka.VelocityPath=0.01; Kuka.CurrentCDSetIndex=0; Kuka.MovementParameterFieldEnabled=True; ArcTech.WdatVarName=WDAT2; ArcTech.Basic=3.4.3.1264
  ;ENDFOLD
  $BWDSTART = FALSE
  LDAT_ACT = LCPDAT2
  FDAT_ACT = FP4
  BAS(#CP_PARAMS, gArcBasVelDefinition)
  SET_CD_PARAMS (0)
  TRIGGER WHEN PATH = ArcGetPath(#ArcOffBefore, WDAT2) DELAY = 0 DO ArcMainNG(#ArcOffBeforeOffStd, WDAT2, WP4) PRIO = -1
  TRIGGER WHEN PATH = ArcGetPath(#OnTheFlyArcOff, WDAT2) DELAY = 0 DO ArcMainNG(#ArcOffMoveStd, WDAT2, WP4) PRIO = -1
  ArcMainNG(#ArcOffBeforeMoveStd, WDAT2, WP4)
  LIN XP4
  ArcMainNG(#ArcOffAfterMoveStd, WDAT2, WP4)
;ENDFOLD
   $VEL.CP = 0.080
   LIN  {X -3.794, Y 4.805, Z 19.300, A 0.000, B 0.000, C 0.000} C_DIS
   $VEL.CP = 0.080
   LIN  {X -4.194, Y 4.205, Z 19.300, A 0.000, B 0.000, C 0.000} C_DIS

;FOLD ARCON WDAT1 LIN P3 Vel=0.5 m/s CPDAT1 Tool[1]:cmttorch Base[1]:vrashatel ;%{PE}
  ;FOLD Parameters ;%{h}
    ;Params IlfProvider=kukaroboter.arctech.arconlin; Kuka.IsGlobalPoint=False; Kuka.PointName=P3; Kuka.BlendingEnabled=False; Kuka.MoveDataName=CPDAT1; Kuka.VelocityPath=0.5; Kuka.CurrentCDSetIndex=0; Kuka.MovementParameterFieldEnabled=True; ArcTech.WdatVarName=WDAT1; ArcTech.Basic=3.4.3.1264
  ;ENDFOLD
  $BWDSTART = FALSE
  LDAT_ACT = LCPDAT1
  FDAT_ACT = FP3
  BAS(#CP_PARAMS, 0.5)
  SET_CD_PARAMS (0)
  TRIGGER WHEN DISTANCE = 1 DELAY = ArcGetDelay(#PreDefinition, WDAT1) DO ArcMainNG(#PreDefinition, WDAT1, WP3) PRIO = -1
  TRIGGER WHEN PATH = ArcGetPath(#OnTheFlyArcOn, WDAT1) DELAY = ArcGetDelay(#GasPreflow, WDAT1) DO ArcMainNG(#GasPreflow, WDAT1, WP3) PRIO = -1
  TRIGGER WHEN PATH = ArcGetPath(#OnTheFlyArcOn, WDAT1) DELAY = 0 DO ArcMainNG(#ArcOnMoveStd, WDAT1, WP3) PRIO = -1
  ArcMainNG(#ArcOnBeforeMoveStd, WDAT1, WP3)
  LIN XP3
  ArcMainNG(#ArcOnAfterMoveStd, WDAT1, WP3)
;ENDFOLD
   $VEL.CP = 0.060
   LIN  {X -4.194, Y 6.918, Z 19.300, A 0.000, B 0.000, C 0.000} C_DIS
   $VEL.CP = 0.060
   LIN  {X 4.527, Y 6.918, Z 19.300, A 0.000, B 0.000, C 0.000} C_DIS
   $VEL.CP = 0.060
   LIN  {X 4.527, Y 5.754, Z 19.300, A 0.000, B 0.000, C 0.000} C_DIS
   $VEL.CP = 0.060
   LIN  {X -0.403, Y -3.880, Z 19.300, A 0.000, B 0.000, C 0.000} C_DIS
   $VEL.CP = 0.060
   LIN  {X 4.712, Y -3.880, Z 19.300, A 0.000, B 0.000, C 0.000} C_DIS
   $VEL.CP = 0.060
   LIN  {X 4.712, Y -6.593, Z 19.300, A 0.000, B 0.000, C 0.000} C_DIS
   $VEL.CP = 0.060
   LIN  {X -4.278, Y -6.593, Z 19.300, A 0.000, B 0.000, C 0.000} C_DIS
   $VEL.CP = 0.060
   LIN  {X -4.278, Y -5.429, Z 19.300, A 0.000, B 0.000, C 0.000} C_DIS
   $VEL.CP = 0.060
   LIN  {X 0.637, Y 4.205, Z 19.300, A 0.000, B 0.000, C 0.000} C_DIS
   $VEL.CP = 0.060
   LIN  {X -4.194, Y 4.205, Z 19.300, A 0.000, B 0.000, C 0.000} C_DIS

;FOLD ARCOFF WDAT2 LIN P4 CPDAT2 Tool[1]:cmttorch Base[1]:vrashatel ;%{PE}
  ;FOLD Parameters ;%{h}
    ;Params IlfProvider=kukaroboter.arctech.arcofflin; Kuka.IsGlobalPoint=False; Kuka.PointName=P4; Kuka.BlendingEnabled=False; Kuka.MoveDataName=CPDAT2; Kuka.VelocityPath=0.01; Kuka.CurrentCDSetIndex=0; Kuka.MovementParameterFieldEnabled=True; ArcTech.WdatVarName=WDAT2; ArcTech.Basic=3.4.3.1264
  ;ENDFOLD
  $BWDSTART = FALSE
  LDAT_ACT = LCPDAT2
  FDAT_ACT = FP4
  BAS(#CP_PARAMS, gArcBasVelDefinition)
  SET_CD_PARAMS (0)
  TRIGGER WHEN PATH = ArcGetPath(#ArcOffBefore, WDAT2) DELAY = 0 DO ArcMainNG(#ArcOffBeforeOffStd, WDAT2, WP4) PRIO = -1
  TRIGGER WHEN PATH = ArcGetPath(#OnTheFlyArcOff, WDAT2) DELAY = 0 DO ArcMainNG(#ArcOffMoveStd, WDAT2, WP4) PRIO = -1
  ArcMainNG(#ArcOffBeforeMoveStd, WDAT2, WP4)
  LIN XP4
  ArcMainNG(#ArcOffAfterMoveStd, WDAT2, WP4)
;ENDFOLD
   $VEL.CP = 0.080
   LIN  {X -4.390, Y 7.114, Z 19.300, A 0.000, B 0.000, C 0.000} C_DIS
   $VEL.CP = 0.080
   LIN  {X -4.390, Y 9.190, Z 19.300, A 0.000, B 0.000, C 0.000} C_DIS
   $VEL.CP = 0.080
   LIN  {X -9.400, Y 9.400, Z 19.300, A 0.000, B 0.000, C 0.000} C_DIS

;FOLD ARCON WDAT1 LIN P3 Vel=0.5 m/s CPDAT1 Tool[1]:cmttorch Base[1]:vrashatel ;%{PE}
  ;FOLD Parameters ;%{h}
    ;Params IlfProvider=kukaroboter.arctech.arconlin; Kuka.IsGlobalPoint=False; Kuka.PointName=P3; Kuka.BlendingEnabled=False; Kuka.MoveDataName=CPDAT1; Kuka.VelocityPath=0.5; Kuka.CurrentCDSetIndex=0; Kuka.MovementParameterFieldEnabled=True; ArcTech.WdatVarName=WDAT1; ArcTech.Basic=3.4.3.1264
  ;ENDFOLD
  $BWDSTART = FALSE
  LDAT_ACT = LCPDAT1
  FDAT_ACT = FP3
  BAS(#CP_PARAMS, 0.5)
  SET_CD_PARAMS (0)
  TRIGGER WHEN DISTANCE = 1 DELAY = ArcGetDelay(#PreDefinition, WDAT1) DO ArcMainNG(#PreDefinition, WDAT1, WP3) PRIO = -1
  TRIGGER WHEN PATH = ArcGetPath(#OnTheFlyArcOn, WDAT1) DELAY = ArcGetDelay(#GasPreflow, WDAT1) DO ArcMainNG(#GasPreflow, WDAT1, WP3) PRIO = -1
  TRIGGER WHEN PATH = ArcGetPath(#OnTheFlyArcOn, WDAT1) DELAY = 0 DO ArcMainNG(#ArcOnMoveStd, WDAT1, WP3) PRIO = -1
  ArcMainNG(#ArcOnBeforeMoveStd, WDAT1, WP3)
  LIN XP3
  ArcMainNG(#ArcOnAfterMoveStd, WDAT1, WP3)
;ENDFOLD
   $VEL.CP = 0.025
   LIN  {X -9.400, Y 9.400, Z 19.300, A 0.000, B 0.000, C 0.000} C_DIS
   $VEL.CP = 0.060
   LIN  {X -9.400, Y -9.400, Z 19.300, A 0.000, B 0.000, C 0.000} C_DIS
   $VEL.CP = 0.060
   LIN  {X 9.400, Y -9.400, Z 19.300, A 0.000, B 0.000, C 0.000} C_DIS
   $VEL.CP = 0.060
   LIN  {X 9.400, Y 9.400, Z 19.300, A 0.000, B 0.000, C 0.000} C_DIS
   $VEL.CP = 0.060
   LIN  {X -9.400, Y 9.400, Z 19.300, A 0.000, B 0.000, C 0.000} C_DIS

;FOLD ARCOFF WDAT2 LIN P4 CPDAT2 Tool[1]:cmttorch Base[1]:vrashatel ;%{PE}
  ;FOLD Parameters ;%{h}
    ;Params IlfProvider=kukaroboter.arctech.arcofflin; Kuka.IsGlobalPoint=False; Kuka.PointName=P4; Kuka.BlendingEnabled=False; Kuka.MoveDataName=CPDAT2; Kuka.VelocityPath=0.01; Kuka.CurrentCDSetIndex=0; Kuka.MovementParameterFieldEnabled=True; ArcTech.WdatVarName=WDAT2; ArcTech.Basic=3.4.3.1264
  ;ENDFOLD
  $BWDSTART = FALSE
  LDAT_ACT = LCPDAT2
  FDAT_ACT = FP4
  BAS(#CP_PARAMS, gArcBasVelDefinition)
  SET_CD_PARAMS (0)
  TRIGGER WHEN PATH = ArcGetPath(#ArcOffBefore, WDAT2) DELAY = 0 DO ArcMainNG(#ArcOffBeforeOffStd, WDAT2, WP4) PRIO = -1
  TRIGGER WHEN PATH = ArcGetPath(#OnTheFlyArcOff, WDAT2) DELAY = 0 DO ArcMainNG(#ArcOffMoveStd, WDAT2, WP4) PRIO = -1
  ArcMainNG(#ArcOffBeforeMoveStd, WDAT2, WP4)
  LIN XP4
  ArcMainNG(#ArcOffAfterMoveStd, WDAT2, WP4)
;ENDFOLD
   $VEL.CP = 0.080
   LIN  {X -9.010, Y 9.010, Z 19.300, A 0.000, B 0.000, C 0.000} C_DIS

;FOLD ARCON WDAT1 LIN P3 Vel=0.5 m/s CPDAT1 Tool[1]:cmttorch Base[1]:vrashatel ;%{PE}
  ;FOLD Parameters ;%{h}
    ;Params IlfProvider=kukaroboter.arctech.arconlin; Kuka.IsGlobalPoint=False; Kuka.PointName=P3; Kuka.BlendingEnabled=False; Kuka.MoveDataName=CPDAT1; Kuka.VelocityPath=0.5; Kuka.CurrentCDSetIndex=0; Kuka.MovementParameterFieldEnabled=True; ArcTech.WdatVarName=WDAT1; ArcTech.Basic=3.4.3.1264
  ;ENDFOLD
  $BWDSTART = FALSE
  LDAT_ACT = LCPDAT1
  FDAT_ACT = FP3
  BAS(#CP_PARAMS, 0.5)
  SET_CD_PARAMS (0)
  TRIGGER WHEN DISTANCE = 1 DELAY = ArcGetDelay(#PreDefinition, WDAT1) DO ArcMainNG(#PreDefinition, WDAT1, WP3) PRIO = -1
  TRIGGER WHEN PATH = ArcGetPath(#OnTheFlyArcOn, WDAT1) DELAY = ArcGetDelay(#GasPreflow, WDAT1) DO ArcMainNG(#GasPreflow, WDAT1, WP3) PRIO = -1
  TRIGGER WHEN PATH = ArcGetPath(#OnTheFlyArcOn, WDAT1) DELAY = 0 DO ArcMainNG(#ArcOnMoveStd, WDAT1, WP3) PRIO = -1
  ArcMainNG(#ArcOnBeforeMoveStd, WDAT1, WP3)
  LIN XP3
  ArcMainNG(#ArcOnAfterMoveStd, WDAT1, WP3)
;ENDFOLD
   $VEL.CP = 0.060
   LIN  {X -9.010, Y -9.010, Z 19.300, A 0.000, B 0.000, C 0.000} C_DIS
   $VEL.CP = 0.060
   LIN  {X 9.010, Y -9.010, Z 19.300, A 0.000, B 0.000, C 0.000} C_DIS
   $VEL.CP = 0.060
   LIN  {X 9.010, Y 9.010, Z 19.300, A 0.000, B 0.000, C 0.000} C_DIS
   $VEL.CP = 0.060
   LIN  {X -9.010, Y 9.010, Z 19.300, A 0.000, B 0.000, C 0.000} C_DIS

;FOLD ARCOFF WDAT2 LIN P4 CPDAT2 Tool[1]:cmttorch Base[1]:vrashatel ;%{PE}
  ;FOLD Parameters ;%{h}
    ;Params IlfProvider=kukaroboter.arctech.arcofflin; Kuka.IsGlobalPoint=False; Kuka.PointName=P4; Kuka.BlendingEnabled=False; Kuka.MoveDataName=CPDAT2; Kuka.VelocityPath=0.01; Kuka.CurrentCDSetIndex=0; Kuka.MovementParameterFieldEnabled=True; ArcTech.WdatVarName=WDAT2; ArcTech.Basic=3.4.3.1264
  ;ENDFOLD
  $BWDSTART = FALSE
  LDAT_ACT = LCPDAT2
  FDAT_ACT = FP4
  BAS(#CP_PARAMS, gArcBasVelDefinition)
  SET_CD_PARAMS (0)
  TRIGGER WHEN PATH = ArcGetPath(#ArcOffBefore, WDAT2) DELAY = 0 DO ArcMainNG(#ArcOffBeforeOffStd, WDAT2, WP4) PRIO = -1
  TRIGGER WHEN PATH = ArcGetPath(#OnTheFlyArcOff, WDAT2) DELAY = 0 DO ArcMainNG(#ArcOffMoveStd, WDAT2, WP4) PRIO = -1
  ArcMainNG(#ArcOffBeforeMoveStd, WDAT2, WP4)
  LIN XP4
  ArcMainNG(#ArcOffAfterMoveStd, WDAT2, WP4)
;ENDFOLD
   $VEL.CP = 0.080
   LIN  {X -9.290, Y 9.010, Z 19.300, A 0.000, B 0.000, C 0.000} C_DIS
   $VEL.CP = 0.080
   LIN  {X -9.218, Y 9.218, Z 19.300, A 0.000, B 0.000, C 0.000} C_DIS
   $VEL.CP = 0.080
   LIN  {X -4.304, Y 9.190, Z 19.300, A 0.000, B 0.000, C 0.000} C_DIS
   $VEL.CP = 0.080
   LIN  {X -4.304, Y 7.108, Z 19.300, A 0.000, B 0.000, C 0.000} C_DIS
   $VEL.CP = 0.080
   LIN  {X -4.584, Y 7.308, Z 19.300, A 0.000, B 0.000, C 0.000} C_DIS

;FOLD ARCON WDAT1 LIN P3 Vel=0.5 m/s CPDAT1 Tool[1]:cmttorch Base[1]:vrashatel ;%{PE}
  ;FOLD Parameters ;%{h}
    ;Params IlfProvider=kukaroboter.arctech.arconlin; Kuka.IsGlobalPoint=False; Kuka.PointName=P3; Kuka.BlendingEnabled=False; Kuka.MoveDataName=CPDAT1; Kuka.VelocityPath=0.5; Kuka.CurrentCDSetIndex=0; Kuka.MovementParameterFieldEnabled=True; ArcTech.WdatVarName=WDAT1; ArcTech.Basic=3.4.3.1264
  ;ENDFOLD
  $BWDSTART = FALSE
  LDAT_ACT = LCPDAT1
  FDAT_ACT = FP3
  BAS(#CP_PARAMS, 0.5)
  SET_CD_PARAMS (0)
  TRIGGER WHEN DISTANCE = 1 DELAY = ArcGetDelay(#PreDefinition, WDAT1) DO ArcMainNG(#PreDefinition, WDAT1, WP3) PRIO = -1
  TRIGGER WHEN PATH = ArcGetPath(#OnTheFlyArcOn, WDAT1) DELAY = ArcGetDelay(#GasPreflow, WDAT1) DO ArcMainNG(#GasPreflow, WDAT1, WP3) PRIO = -1
  TRIGGER WHEN PATH = ArcGetPath(#OnTheFlyArcOn, WDAT1) DELAY = 0 DO ArcMainNG(#ArcOnMoveStd, WDAT1, WP3) PRIO = -1
  ArcMainNG(#ArcOnBeforeMoveStd, WDAT1, WP3)
  LIN XP3
  ArcMainNG(#ArcOnAfterMoveStd, WDAT1, WP3)
;ENDFOLD
   $VEL.CP = 0.025
   LIN  {X -4.584, Y 7.308, Z 19.300, A 0.000, B 0.000, C 0.000} C_DIS
   $VEL.CP = 0.060
   LIN  {X 4.917, Y 7.308, Z 19.300, A 0.000, B 0.000, C 0.000} C_DIS
   $VEL.CP = 0.060
   LIN  {X 4.917, Y 5.660, Z 19.300, A 0.000, B 0.000, C 0.000} C_DIS
   $VEL.CP = 0.060
   LIN  {X 0.235, Y -3.490, Z 19.300, A 0.000, B 0.000, C 0.000} C_DIS
   $VEL.CP = 0.060
   LIN  {X 5.102, Y -3.490, Z 19.300, A 0.000, B 0.000, C 0.000} C_DIS
   $VEL.CP = 0.060
   LIN  {X 5.102, Y -6.983, Z 19.300, A 0.000, B 0.000, C 0.000} C_DIS
   $VEL.CP = 0.060
   LIN  {X -4.668, Y -6.983, Z 19.300, A 0.000, B 0.000, C 0.000} C_DIS
   $VEL.CP = 0.060
   LIN  {X -4.668, Y -5.335, Z 19.300, A 0.000, B 0.000, C 0.000} C_DIS
   $VEL.CP = 0.060
   LIN  {X 0.001, Y 3.815, Z 19.300, A 0.000, B 0.000, C 0.000} C_DIS
   $VEL.CP = 0.060
   LIN  {X -4.584, Y 3.815, Z 19.300, A 0.000, B 0.000, C 0.000} C_DIS
   $VEL.CP = 0.060
   LIN  {X -4.584, Y 7.308, Z 19.300, A 0.000, B 0.000, C 0.000} C_DIS

;FOLD ARCOFF WDAT2 LIN P4 CPDAT2 Tool[1]:cmttorch Base[1]:vrashatel ;%{PE}
  ;FOLD Parameters ;%{h}
    ;Params IlfProvider=kukaroboter.arctech.arcofflin; Kuka.IsGlobalPoint=False; Kuka.PointName=P4; Kuka.BlendingEnabled=False; Kuka.MoveDataName=CPDAT2; Kuka.VelocityPath=0.01; Kuka.CurrentCDSetIndex=0; Kuka.MovementParameterFieldEnabled=True; ArcTech.WdatVarName=WDAT2; ArcTech.Basic=3.4.3.1264
  ;ENDFOLD
  $BWDSTART = FALSE
  LDAT_ACT = LCPDAT2
  FDAT_ACT = FP4
  BAS(#CP_PARAMS, gArcBasVelDefinition)
  SET_CD_PARAMS (0)
  TRIGGER WHEN PATH = ArcGetPath(#ArcOffBefore, WDAT2) DELAY = 0 DO ArcMainNG(#ArcOffBeforeOffStd, WDAT2, WP4) PRIO = -1
  TRIGGER WHEN PATH = ArcGetPath(#OnTheFlyArcOff, WDAT2) DELAY = 0 DO ArcMainNG(#ArcOffMoveStd, WDAT2, WP4) PRIO = -1
  ArcMainNG(#ArcOffBeforeMoveStd, WDAT2, WP4)
  LIN XP4
  ArcMainNG(#ArcOffAfterMoveStd, WDAT2, WP4)
;ENDFOLD
   $VEL.CP = 0.080
   LIN  {X -4.304, Y 7.058, Z 19.300, A 0.000, B 0.000, C 0.000} C_DIS
   $VEL.CP = 0.080
   LIN  {X 4.723, Y 7.114, Z 19.300, A 0.000, B 0.000, C 0.000} C_DIS
   $VEL.CP = 0.080
   LIN  {X 4.723, Y 9.190, Z 19.300, A 0.000, B 0.000, C 0.000} C_DIS
   $VEL.CP = 0.080
   LIN  {X 8.706, Y 9.290, Z 19.300, A 0.000, B 0.000, C 0.000} C_DIS
   $VEL.CP = 0.080
   LIN  {X 8.706, Y 8.829, Z 19.300, A 0.000, B 0.000, C 0.000} C_DIS

;FOLD ARCON WDAT1 LIN P3 Vel=0.5 m/s CPDAT1 Tool[1]:cmttorch Base[1]:vrashatel ;%{PE}
  ;FOLD Parameters ;%{h}
    ;Params IlfProvider=kukaroboter.arctech.arconlin; Kuka.IsGlobalPoint=False; Kuka.PointName=P3; Kuka.BlendingEnabled=False; Kuka.MoveDataName=CPDAT1; Kuka.VelocityPath=0.5; Kuka.CurrentCDSetIndex=0; Kuka.MovementParameterFieldEnabled=True; ArcTech.WdatVarName=WDAT1; ArcTech.Basic=3.4.3.1264
  ;ENDFOLD
  $BWDSTART = FALSE
  LDAT_ACT = LCPDAT1
  FDAT_ACT = FP3
  BAS(#CP_PARAMS, 0.5)
  SET_CD_PARAMS (0)
  TRIGGER WHEN DISTANCE = 1 DELAY = ArcGetDelay(#PreDefinition, WDAT1) DO ArcMainNG(#PreDefinition, WDAT1, WP3) PRIO = -1
  TRIGGER WHEN PATH = ArcGetPath(#OnTheFlyArcOn, WDAT1) DELAY = ArcGetDelay(#GasPreflow, WDAT1) DO ArcMainNG(#GasPreflow, WDAT1, WP3) PRIO = -1
  TRIGGER WHEN PATH = ArcGetPath(#OnTheFlyArcOn, WDAT1) DELAY = 0 DO ArcMainNG(#ArcOnMoveStd, WDAT1, WP3) PRIO = -1
  ArcMainNG(#ArcOnBeforeMoveStd, WDAT1, WP3)
  LIN XP3
  ArcMainNG(#ArcOnAfterMoveStd, WDAT1, WP3)
;ENDFOLD
   $VEL.CP = 0.025
   LIN  {X 8.706, Y 8.829, Z 19.300, A 0.000, B 0.000, C 0.000} C_DIS
   $VEL.CP = 0.060
   LIN  {X 8.829, Y 8.706, Z 19.300, A 0.000, B 0.000, C 0.000} C_DIS

;FOLD ARCOFF WDAT2 LIN P4 CPDAT2 Tool[1]:cmttorch Base[1]:vrashatel ;%{PE}
  ;FOLD Parameters ;%{h}
    ;Params IlfProvider=kukaroboter.arctech.arcofflin; Kuka.IsGlobalPoint=False; Kuka.PointName=P4; Kuka.BlendingEnabled=False; Kuka.MoveDataName=CPDAT2; Kuka.VelocityPath=0.01; Kuka.CurrentCDSetIndex=0; Kuka.MovementParameterFieldEnabled=True; ArcTech.WdatVarName=WDAT2; ArcTech.Basic=3.4.3.1264
  ;ENDFOLD
  $BWDSTART = FALSE
  LDAT_ACT = LCPDAT2
  FDAT_ACT = FP4
  BAS(#CP_PARAMS, gArcBasVelDefinition)
  SET_CD_PARAMS (0)
  TRIGGER WHEN PATH = ArcGetPath(#ArcOffBefore, WDAT2) DELAY = 0 DO ArcMainNG(#ArcOffBeforeOffStd, WDAT2, WP4) PRIO = -1
  TRIGGER WHEN PATH = ArcGetPath(#OnTheFlyArcOff, WDAT2) DELAY = 0 DO ArcMainNG(#ArcOffMoveStd, WDAT2, WP4) PRIO = -1
  ArcMainNG(#ArcOffBeforeMoveStd, WDAT2, WP4)
  LIN XP4
  ArcMainNG(#ArcOffAfterMoveStd, WDAT2, WP4)
;ENDFOLD
   $VEL.CP = 0.080
   LIN  {X 8.829, Y 8.140, Z 19.300, A 0.000, B 0.000, C 0.000} C_DIS

;FOLD ARCON WDAT1 LIN P3 Vel=0.5 m/s CPDAT1 Tool[1]:cmttorch Base[1]:vrashatel ;%{PE}
  ;FOLD Parameters ;%{h}
    ;Params IlfProvider=kukaroboter.arctech.arconlin; Kuka.IsGlobalPoint=False; Kuka.PointName=P3; Kuka.BlendingEnabled=False; Kuka.MoveDataName=CPDAT1; Kuka.VelocityPath=0.5; Kuka.CurrentCDSetIndex=0; Kuka.MovementParameterFieldEnabled=True; ArcTech.WdatVarName=WDAT1; ArcTech.Basic=3.4.3.1264
  ;ENDFOLD
  $BWDSTART = FALSE
  LDAT_ACT = LCPDAT1
  FDAT_ACT = FP3
  BAS(#CP_PARAMS, 0.5)
  SET_CD_PARAMS (0)
  TRIGGER WHEN DISTANCE = 1 DELAY = ArcGetDelay(#PreDefinition, WDAT1) DO ArcMainNG(#PreDefinition, WDAT1, WP3) PRIO = -1
  TRIGGER WHEN PATH = ArcGetPath(#OnTheFlyArcOn, WDAT1) DELAY = ArcGetDelay(#GasPreflow, WDAT1) DO ArcMainNG(#GasPreflow, WDAT1, WP3) PRIO = -1
  TRIGGER WHEN PATH = ArcGetPath(#OnTheFlyArcOn, WDAT1) DELAY = 0 DO ArcMainNG(#ArcOnMoveStd, WDAT1, WP3) PRIO = -1
  ArcMainNG(#ArcOnBeforeMoveStd, WDAT1, WP3)
  LIN XP3
  ArcMainNG(#ArcOnAfterMoveStd, WDAT1, WP3)
;ENDFOLD
   $VEL.CP = 0.060
   LIN  {X 8.140, Y 8.829, Z 19.300, A 0.000, B 0.000, C 0.000} C_DIS

;FOLD ARCOFF WDAT2 LIN P4 CPDAT2 Tool[1]:cmttorch Base[1]:vrashatel ;%{PE}
  ;FOLD Parameters ;%{h}
    ;Params IlfProvider=kukaroboter.arctech.arcofflin; Kuka.IsGlobalPoint=False; Kuka.PointName=P4; Kuka.BlendingEnabled=False; Kuka.MoveDataName=CPDAT2; Kuka.VelocityPath=0.01; Kuka.CurrentCDSetIndex=0; Kuka.MovementParameterFieldEnabled=True; ArcTech.WdatVarName=WDAT2; ArcTech.Basic=3.4.3.1264
  ;ENDFOLD
  $BWDSTART = FALSE
  LDAT_ACT = LCPDAT2
  FDAT_ACT = FP4
  BAS(#CP_PARAMS, gArcBasVelDefinition)
  SET_CD_PARAMS (0)
  TRIGGER WHEN PATH = ArcGetPath(#ArcOffBefore, WDAT2) DELAY = 0 DO ArcMainNG(#ArcOffBeforeOffStd, WDAT2, WP4) PRIO = -1
  TRIGGER WHEN PATH = ArcGetPath(#OnTheFlyArcOff, WDAT2) DELAY = 0 DO ArcMainNG(#ArcOffMoveStd, WDAT2, WP4) PRIO = -1
  ArcMainNG(#ArcOffBeforeMoveStd, WDAT2, WP4)
  LIN XP4
  ArcMainNG(#ArcOffAfterMoveStd, WDAT2, WP4)
;ENDFOLD
   $VEL.CP = 0.080
   LIN  {X 7.575, Y 8.829, Z 19.300, A 0.000, B 0.000, C 0.000} C_DIS

;FOLD ARCON WDAT1 LIN P3 Vel=0.5 m/s CPDAT1 Tool[1]:cmttorch Base[1]:vrashatel ;%{PE}
  ;FOLD Parameters ;%{h}
    ;Params IlfProvider=kukaroboter.arctech.arconlin; Kuka.IsGlobalPoint=False; Kuka.PointName=P3; Kuka.BlendingEnabled=False; Kuka.MoveDataName=CPDAT1; Kuka.VelocityPath=0.5; Kuka.CurrentCDSetIndex=0; Kuka.MovementParameterFieldEnabled=True; ArcTech.WdatVarName=WDAT1; ArcTech.Basic=3.4.3.1264
  ;ENDFOLD
  $BWDSTART = FALSE
  LDAT_ACT = LCPDAT1
  FDAT_ACT = FP3
  BAS(#CP_PARAMS, 0.5)
  SET_CD_PARAMS (0)
  TRIGGER WHEN DISTANCE = 1 DELAY = ArcGetDelay(#PreDefinition, WDAT1) DO ArcMainNG(#PreDefinition, WDAT1, WP3) PRIO = -1
  TRIGGER WHEN PATH = ArcGetPath(#OnTheFlyArcOn, WDAT1) DELAY = ArcGetDelay(#GasPreflow, WDAT1) DO ArcMainNG(#GasPreflow, WDAT1, WP3) PRIO = -1
  TRIGGER WHEN PATH = ArcGetPath(#OnTheFlyArcOn, WDAT1) DELAY = 0 DO ArcMainNG(#ArcOnMoveStd, WDAT1, WP3) PRIO = -1
  ArcMainNG(#ArcOnBeforeMoveStd, WDAT1, WP3)
  LIN XP3
  ArcMainNG(#ArcOnAfterMoveStd, WDAT1, WP3)
;ENDFOLD
   $VEL.CP = 0.060
   LIN  {X 8.829, Y 7.575, Z 19.300, A 0.000, B 0.000, C 0.000} C_DIS

;FOLD ARCOFF WDAT2 LIN P4 CPDAT2 Tool[1]:cmttorch Base[1]:vrashatel ;%{PE}
  ;FOLD Parameters ;%{h}
    ;Params IlfProvider=kukaroboter.arctech.arcofflin; Kuka.IsGlobalPoint=False; Kuka.PointName=P4; Kuka.BlendingEnabled=False; Kuka.MoveDataName=CPDAT2; Kuka.VelocityPath=0.01; Kuka.CurrentCDSetIndex=0; Kuka.MovementParameterFieldEnabled=True; ArcTech.WdatVarName=WDAT2; ArcTech.Basic=3.4.3.1264
  ;ENDFOLD
  $BWDSTART = FALSE
  LDAT_ACT = LCPDAT2
  FDAT_ACT = FP4
  BAS(#CP_PARAMS, gArcBasVelDefinition)
  SET_CD_PARAMS (0)
  TRIGGER WHEN PATH = ArcGetPath(#ArcOffBefore, WDAT2) DELAY = 0 DO ArcMainNG(#ArcOffBeforeOffStd, WDAT2, WP4) PRIO = -1
  TRIGGER WHEN PATH = ArcGetPath(#OnTheFlyArcOff, WDAT2) DELAY = 0 DO ArcMainNG(#ArcOffMoveStd, WDAT2, WP4) PRIO = -1
  ArcMainNG(#ArcOffBeforeMoveStd, WDAT2, WP4)
  LIN XP4
  ArcMainNG(#ArcOffAfterMoveStd, WDAT2, WP4)
;ENDFOLD
   $VEL.CP = 0.080
   LIN  {X 8.829, Y 7.009, Z 19.300, A 0.000, B 0.000, C 0.000} C_DIS

;FOLD ARCON WDAT1 LIN P3 Vel=0.5 m/s CPDAT1 Tool[1]:cmttorch Base[1]:vrashatel ;%{PE}
  ;FOLD Parameters ;%{h}
    ;Params IlfProvider=kukaroboter.arctech.arconlin; Kuka.IsGlobalPoint=False; Kuka.PointName=P3; Kuka.BlendingEnabled=False; Kuka.MoveDataName=CPDAT1; Kuka.VelocityPath=0.5; Kuka.CurrentCDSetIndex=0; Kuka.MovementParameterFieldEnabled=True; ArcTech.WdatVarName=WDAT1; ArcTech.Basic=3.4.3.1264
  ;ENDFOLD
  $BWDSTART = FALSE
  LDAT_ACT = LCPDAT1
  FDAT_ACT = FP3
  BAS(#CP_PARAMS, 0.5)
  SET_CD_PARAMS (0)
  TRIGGER WHEN DISTANCE = 1 DELAY = ArcGetDelay(#PreDefinition, WDAT1) DO ArcMainNG(#PreDefinition, WDAT1, WP3) PRIO = -1
  TRIGGER WHEN PATH = ArcGetPath(#OnTheFlyArcOn, WDAT1) DELAY = ArcGetDelay(#GasPreflow, WDAT1) DO ArcMainNG(#GasPreflow, WDAT1, WP3) PRIO = -1
  TRIGGER WHEN PATH = ArcGetPath(#OnTheFlyArcOn, WDAT1) DELAY = 0 DO ArcMainNG(#ArcOnMoveStd, WDAT1, WP3) PRIO = -1
  ArcMainNG(#ArcOnBeforeMoveStd, WDAT1, WP3)
  LIN XP3
  ArcMainNG(#ArcOnAfterMoveStd, WDAT1, WP3)
;ENDFOLD
   $VEL.CP = 0.060
   LIN  {X 7.009, Y 8.829, Z 19.300, A 0.000, B 0.000, C 0.000} C_DIS

;FOLD ARCOFF WDAT2 LIN P4 CPDAT2 Tool[1]:cmttorch Base[1]:vrashatel ;%{PE}
  ;FOLD Parameters ;%{h}
    ;Params IlfProvider=kukaroboter.arctech.arcofflin; Kuka.IsGlobalPoint=False; Kuka.PointName=P4; Kuka.BlendingEnabled=False; Kuka.MoveDataName=CPDAT2; Kuka.VelocityPath=0.01; Kuka.CurrentCDSetIndex=0; Kuka.MovementParameterFieldEnabled=True; ArcTech.WdatVarName=WDAT2; ArcTech.Basic=3.4.3.1264
  ;ENDFOLD
  $BWDSTART = FALSE
  LDAT_ACT = LCPDAT2
  FDAT_ACT = FP4
  BAS(#CP_PARAMS, gArcBasVelDefinition)
  SET_CD_PARAMS (0)
  TRIGGER WHEN PATH = ArcGetPath(#ArcOffBefore, WDAT2) DELAY = 0 DO ArcMainNG(#ArcOffBeforeOffStd, WDAT2, WP4) PRIO = -1
  TRIGGER WHEN PATH = ArcGetPath(#OnTheFlyArcOff, WDAT2) DELAY = 0 DO ArcMainNG(#ArcOffMoveStd, WDAT2, WP4) PRIO = -1
  ArcMainNG(#ArcOffBeforeMoveStd, WDAT2, WP4)
  LIN XP4
  ArcMainNG(#ArcOffAfterMoveStd, WDAT2, WP4)
;ENDFOLD
   $VEL.CP = 0.080
   LIN  {X 6.443, Y 8.829, Z 19.300, A 0.000, B 0.000, C 0.000} C_DIS

;FOLD ARCON WDAT1 LIN P3 Vel=0.5 m/s CPDAT1 Tool[1]:cmttorch Base[1]:vrashatel ;%{PE}
  ;FOLD Parameters ;%{h}
    ;Params IlfProvider=kukaroboter.arctech.arconlin; Kuka.IsGlobalPoint=False; Kuka.PointName=P3; Kuka.BlendingEnabled=False; Kuka.MoveDataName=CPDAT1; Kuka.VelocityPath=0.5; Kuka.CurrentCDSetIndex=0; Kuka.MovementParameterFieldEnabled=True; ArcTech.WdatVarName=WDAT1; ArcTech.Basic=3.4.3.1264
  ;ENDFOLD
  $BWDSTART = FALSE
  LDAT_ACT = LCPDAT1
  FDAT_ACT = FP3
  BAS(#CP_PARAMS, 0.5)
  SET_CD_PARAMS (0)
  TRIGGER WHEN DISTANCE = 1 DELAY = ArcGetDelay(#PreDefinition, WDAT1) DO ArcMainNG(#PreDefinition, WDAT1, WP3) PRIO = -1
  TRIGGER WHEN PATH = ArcGetPath(#OnTheFlyArcOn, WDAT1) DELAY = ArcGetDelay(#GasPreflow, WDAT1) DO ArcMainNG(#GasPreflow, WDAT1, WP3) PRIO = -1
  TRIGGER WHEN PATH = ArcGetPath(#OnTheFlyArcOn, WDAT1) DELAY = 0 DO ArcMainNG(#ArcOnMoveStd, WDAT1, WP3) PRIO = -1
  ArcMainNG(#ArcOnBeforeMoveStd, WDAT1, WP3)
  LIN XP3
  ArcMainNG(#ArcOnAfterMoveStd, WDAT1, WP3)
;ENDFOLD
   $VEL.CP = 0.060
   LIN  {X 8.829, Y 6.443, Z 19.300, A 0.000, B 0.000, C 0.000} C_DIS

;FOLD ARCOFF WDAT2 LIN P4 CPDAT2 Tool[1]:cmttorch Base[1]:vrashatel ;%{PE}
  ;FOLD Parameters ;%{h}
    ;Params IlfProvider=kukaroboter.arctech.arcofflin; Kuka.IsGlobalPoint=False; Kuka.PointName=P4; Kuka.BlendingEnabled=False; Kuka.MoveDataName=CPDAT2; Kuka.VelocityPath=0.01; Kuka.CurrentCDSetIndex=0; Kuka.MovementParameterFieldEnabled=True; ArcTech.WdatVarName=WDAT2; ArcTech.Basic=3.4.3.1264
  ;ENDFOLD
  $BWDSTART = FALSE
  LDAT_ACT = LCPDAT2
  FDAT_ACT = FP4
  BAS(#CP_PARAMS, gArcBasVelDefinition)
  SET_CD_PARAMS (0)
  TRIGGER WHEN PATH = ArcGetPath(#ArcOffBefore, WDAT2) DELAY = 0 DO ArcMainNG(#ArcOffBeforeOffStd, WDAT2, WP4) PRIO = -1
  TRIGGER WHEN PATH = ArcGetPath(#OnTheFlyArcOff, WDAT2) DELAY = 0 DO ArcMainNG(#ArcOffMoveStd, WDAT2, WP4) PRIO = -1
  ArcMainNG(#ArcOffBeforeMoveStd, WDAT2, WP4)
  LIN XP4
  ArcMainNG(#ArcOffAfterMoveStd, WDAT2, WP4)
;ENDFOLD
   $VEL.CP = 0.080
   LIN  {X 8.829, Y 5.878, Z 19.300, A 0.000, B 0.000, C 0.000} C_DIS

;FOLD ARCON WDAT1 LIN P3 Vel=0.5 m/s CPDAT1 Tool[1]:cmttorch Base[1]:vrashatel ;%{PE}
  ;FOLD Parameters ;%{h}
    ;Params IlfProvider=kukaroboter.arctech.arconlin; Kuka.IsGlobalPoint=False; Kuka.PointName=P3; Kuka.BlendingEnabled=False; Kuka.MoveDataName=CPDAT1; Kuka.VelocityPath=0.5; Kuka.CurrentCDSetIndex=0; Kuka.MovementParameterFieldEnabled=True; ArcTech.WdatVarName=WDAT1; ArcTech.Basic=3.4.3.1264
  ;ENDFOLD
  $BWDSTART = FALSE
  LDAT_ACT = LCPDAT1
  FDAT_ACT = FP3
  BAS(#CP_PARAMS, 0.5)
  SET_CD_PARAMS (0)
  TRIGGER WHEN DISTANCE = 1 DELAY = ArcGetDelay(#PreDefinition, WDAT1) DO ArcMainNG(#PreDefinition, WDAT1, WP3) PRIO = -1
  TRIGGER WHEN PATH = ArcGetPath(#OnTheFlyArcOn, WDAT1) DELAY = ArcGetDelay(#GasPreflow, WDAT1) DO ArcMainNG(#GasPreflow, WDAT1, WP3) PRIO = -1
  TRIGGER WHEN PATH = ArcGetPath(#OnTheFlyArcOn, WDAT1) DELAY = 0 DO ArcMainNG(#ArcOnMoveStd, WDAT1, WP3) PRIO = -1
  ArcMainNG(#ArcOnBeforeMoveStd, WDAT1, WP3)
  LIN XP3
  ArcMainNG(#ArcOnAfterMoveStd, WDAT1, WP3)
;ENDFOLD
   $VEL.CP = 0.060
   LIN  {X 5.878, Y 8.829, Z 19.300, A 0.000, B 0.000, C 0.000} C_DIS

;FOLD ARCOFF WDAT2 LIN P4 CPDAT2 Tool[1]:cmttorch Base[1]:vrashatel ;%{PE}
  ;FOLD Parameters ;%{h}
    ;Params IlfProvider=kukaroboter.arctech.arcofflin; Kuka.IsGlobalPoint=False; Kuka.PointName=P4; Kuka.BlendingEnabled=False; Kuka.MoveDataName=CPDAT2; Kuka.VelocityPath=0.01; Kuka.CurrentCDSetIndex=0; Kuka.MovementParameterFieldEnabled=True; ArcTech.WdatVarName=WDAT2; ArcTech.Basic=3.4.3.1264
  ;ENDFOLD
  $BWDSTART = FALSE
  LDAT_ACT = LCPDAT2
  FDAT_ACT = FP4
  BAS(#CP_PARAMS, gArcBasVelDefinition)
  SET_CD_PARAMS (0)
  TRIGGER WHEN PATH = ArcGetPath(#ArcOffBefore, WDAT2) DELAY = 0 DO ArcMainNG(#ArcOffBeforeOffStd, WDAT2, WP4) PRIO = -1
  TRIGGER WHEN PATH = ArcGetPath(#OnTheFlyArcOff, WDAT2) DELAY = 0 DO ArcMainNG(#ArcOffMoveStd, WDAT2, WP4) PRIO = -1
  ArcMainNG(#ArcOffBeforeMoveStd, WDAT2, WP4)
  LIN XP4
  ArcMainNG(#ArcOffAfterMoveStd, WDAT2, WP4)
;ENDFOLD
   $VEL.CP = 0.080
   LIN  {X 5.312, Y 8.829, Z 19.300, A 0.000, B 0.000, C 0.000} C_DIS

;FOLD ARCON WDAT1 LIN P3 Vel=0.5 m/s CPDAT1 Tool[1]:cmttorch Base[1]:vrashatel ;%{PE}
  ;FOLD Parameters ;%{h}
    ;Params IlfProvider=kukaroboter.arctech.arconlin; Kuka.IsGlobalPoint=False; Kuka.PointName=P3; Kuka.BlendingEnabled=False; Kuka.MoveDataName=CPDAT1; Kuka.VelocityPath=0.5; Kuka.CurrentCDSetIndex=0; Kuka.MovementParameterFieldEnabled=True; ArcTech.WdatVarName=WDAT1; ArcTech.Basic=3.4.3.1264
  ;ENDFOLD
  $BWDSTART = FALSE
  LDAT_ACT = LCPDAT1
  FDAT_ACT = FP3
  BAS(#CP_PARAMS, 0.5)
  SET_CD_PARAMS (0)
  TRIGGER WHEN DISTANCE = 1 DELAY = ArcGetDelay(#PreDefinition, WDAT1) DO ArcMainNG(#PreDefinition, WDAT1, WP3) PRIO = -1
  TRIGGER WHEN PATH = ArcGetPath(#OnTheFlyArcOn, WDAT1) DELAY = ArcGetDelay(#GasPreflow, WDAT1) DO ArcMainNG(#GasPreflow, WDAT1, WP3) PRIO = -1
  TRIGGER WHEN PATH = ArcGetPath(#OnTheFlyArcOn, WDAT1) DELAY = 0 DO ArcMainNG(#ArcOnMoveStd, WDAT1, WP3) PRIO = -1
  ArcMainNG(#ArcOnBeforeMoveStd, WDAT1, WP3)
  LIN XP3
  ArcMainNG(#ArcOnAfterMoveStd, WDAT1, WP3)
;ENDFOLD
   $VEL.CP = 0.060
   LIN  {X 8.829, Y 5.312, Z 19.300, A 0.000, B 0.000, C 0.000} C_DIS

;FOLD ARCOFF WDAT2 LIN P4 CPDAT2 Tool[1]:cmttorch Base[1]:vrashatel ;%{PE}
  ;FOLD Parameters ;%{h}
    ;Params IlfProvider=kukaroboter.arctech.arcofflin; Kuka.IsGlobalPoint=False; Kuka.PointName=P4; Kuka.BlendingEnabled=False; Kuka.MoveDataName=CPDAT2; Kuka.VelocityPath=0.01; Kuka.CurrentCDSetIndex=0; Kuka.MovementParameterFieldEnabled=True; ArcTech.WdatVarName=WDAT2; ArcTech.Basic=3.4.3.1264
  ;ENDFOLD
  $BWDSTART = FALSE
  LDAT_ACT = LCPDAT2
  FDAT_ACT = FP4
  BAS(#CP_PARAMS, gArcBasVelDefinition)
  SET_CD_PARAMS (0)
  TRIGGER WHEN PATH = ArcGetPath(#ArcOffBefore, WDAT2) DELAY = 0 DO ArcMainNG(#ArcOffBeforeOffStd, WDAT2, WP4) PRIO = -1
  TRIGGER WHEN PATH = ArcGetPath(#OnTheFlyArcOff, WDAT2) DELAY = 0 DO ArcMainNG(#ArcOffMoveStd, WDAT2, WP4) PRIO = -1
  ArcMainNG(#ArcOffBeforeMoveStd, WDAT2, WP4)
  LIN XP4
  ArcMainNG(#ArcOffAfterMoveStd, WDAT2, WP4)
;ENDFOLD
   $VEL.CP = 0.080
   LIN  {X 8.829, Y 4.746, Z 19.300, A 0.000, B 0.000, C 0.000} C_DIS

;FOLD ARCON WDAT1 LIN P3 Vel=0.5 m/s CPDAT1 Tool[1]:cmttorch Base[1]:vrashatel ;%{PE}
  ;FOLD Parameters ;%{h}
    ;Params IlfProvider=kukaroboter.arctech.arconlin; Kuka.IsGlobalPoint=False; Kuka.PointName=P3; Kuka.BlendingEnabled=False; Kuka.MoveDataName=CPDAT1; Kuka.VelocityPath=0.5; Kuka.CurrentCDSetIndex=0; Kuka.MovementParameterFieldEnabled=True; ArcTech.WdatVarName=WDAT1; ArcTech.Basic=3.4.3.1264
  ;ENDFOLD
  $BWDSTART = FALSE
  LDAT_ACT = LCPDAT1
  FDAT_ACT = FP3
  BAS(#CP_PARAMS, 0.5)
  SET_CD_PARAMS (0)
  TRIGGER WHEN DISTANCE = 1 DELAY = ArcGetDelay(#PreDefinition, WDAT1) DO ArcMainNG(#PreDefinition, WDAT1, WP3) PRIO = -1
  TRIGGER WHEN PATH = ArcGetPath(#OnTheFlyArcOn, WDAT1) DELAY = ArcGetDelay(#GasPreflow, WDAT1) DO ArcMainNG(#GasPreflow, WDAT1, WP3) PRIO = -1
  TRIGGER WHEN PATH = ArcGetPath(#OnTheFlyArcOn, WDAT1) DELAY = 0 DO ArcMainNG(#ArcOnMoveStd, WDAT1, WP3) PRIO = -1
  ArcMainNG(#ArcOnBeforeMoveStd, WDAT1, WP3)
  LIN XP3
  ArcMainNG(#ArcOnAfterMoveStd, WDAT1, WP3)
;ENDFOLD
   $VEL.CP = 0.060
   LIN  {X 4.746, Y 8.829, Z 19.300, A 0.000, B 0.000, C 0.000} C_DIS

;FOLD ARCOFF WDAT2 LIN P4 CPDAT2 Tool[1]:cmttorch Base[1]:vrashatel ;%{PE}
  ;FOLD Parameters ;%{h}
    ;Params IlfProvider=kukaroboter.arctech.arcofflin; Kuka.IsGlobalPoint=False; Kuka.PointName=P4; Kuka.BlendingEnabled=False; Kuka.MoveDataName=CPDAT2; Kuka.VelocityPath=0.01; Kuka.CurrentCDSetIndex=0; Kuka.MovementParameterFieldEnabled=True; ArcTech.WdatVarName=WDAT2; ArcTech.Basic=3.4.3.1264
  ;ENDFOLD
  $BWDSTART = FALSE
  LDAT_ACT = LCPDAT2
  FDAT_ACT = FP4
  BAS(#CP_PARAMS, gArcBasVelDefinition)
  SET_CD_PARAMS (0)
  TRIGGER WHEN PATH = ArcGetPath(#ArcOffBefore, WDAT2) DELAY = 0 DO ArcMainNG(#ArcOffBeforeOffStd, WDAT2, WP4) PRIO = -1
  TRIGGER WHEN PATH = ArcGetPath(#OnTheFlyArcOff, WDAT2) DELAY = 0 DO ArcMainNG(#ArcOffMoveStd, WDAT2, WP4) PRIO = -1
  ArcMainNG(#ArcOffBeforeMoveStd, WDAT2, WP4)
  LIN XP4
  ArcMainNG(#ArcOffAfterMoveStd, WDAT2, WP4)
;ENDFOLD
   $VEL.CP = 0.080
   LIN  {X 4.181, Y 8.829, Z 19.300, A 0.000, B 0.000, C 0.000} C_DIS

;FOLD ARCON WDAT1 LIN P3 Vel=0.5 m/s CPDAT1 Tool[1]:cmttorch Base[1]:vrashatel ;%{PE}
  ;FOLD Parameters ;%{h}
    ;Params IlfProvider=kukaroboter.arctech.arconlin; Kuka.IsGlobalPoint=False; Kuka.PointName=P3; Kuka.BlendingEnabled=False; Kuka.MoveDataName=CPDAT1; Kuka.VelocityPath=0.5; Kuka.CurrentCDSetIndex=0; Kuka.MovementParameterFieldEnabled=True; ArcTech.WdatVarName=WDAT1; ArcTech.Basic=3.4.3.1264
  ;ENDFOLD
  $BWDSTART = FALSE
  LDAT_ACT = LCPDAT1
  FDAT_ACT = FP3
  BAS(#CP_PARAMS, 0.5)
  SET_CD_PARAMS (0)
  TRIGGER WHEN DISTANCE = 1 DELAY = ArcGetDelay(#PreDefinition, WDAT1) DO ArcMainNG(#PreDefinition, WDAT1, WP3) PRIO = -1
  TRIGGER WHEN PATH = ArcGetPath(#OnTheFlyArcOn, WDAT1) DELAY = ArcGetDelay(#GasPreflow, WDAT1) DO ArcMainNG(#GasPreflow, WDAT1, WP3) PRIO = -1
  TRIGGER WHEN PATH = ArcGetPath(#OnTheFlyArcOn, WDAT1) DELAY = 0 DO ArcMainNG(#ArcOnMoveStd, WDAT1, WP3) PRIO = -1
  ArcMainNG(#ArcOnBeforeMoveStd, WDAT1, WP3)
  LIN XP3
  ArcMainNG(#ArcOnAfterMoveStd, WDAT1, WP3)
;ENDFOLD
   $VEL.CP = 0.060
   LIN  {X 8.829, Y 4.181, Z 19.300, A 0.000, B 0.000, C 0.000} C_DIS

